C07282=1029.317,321.724,369.650,171.379,46.415,159.024
C07283=1029.324,321.936,369.619,171.383,46.415,159.025
C07284=1029.330,322.147,369.590,171.388,46.415,159.025
C07285=1029.337,322.395,369.555,171.392,46.415,159.026
C07286=1029.345,322.642,369.521,171.398,46.415,159.026
C07287=1029.351,322.890,369.486,171.403,46.416,159.027
C07288=1029.360,323.137,369.451,171.409,46.416,159.028
C07289=1029.366,323.385,369.416,171.414,46.416,159.028
C07290=1029.374,323.632,369.382,171.419,46.416,159.029
C07291=1029.381,323.879,369.348,171.424,46.416,159.030
C07292=1029.388,324.127,369.312,171.429,46.416,159.030
C07293=1029.396,324.375,369.278,171.435,46.417,159.031
C07294=1029.403,324.622,369.243,171.441,46.417,159.032
C07295=1029.410,324.869,369.208,171.445,46.417,159.032
C07296=1029.418,325.117,369.173,171.451,46.417,159.033
C07297=1029.425,325.364,369.138,171.457,46.417,159.034
C07298=1029.433,325.611,369.104,171.461,46.417,159.034
C07299=1029.440,325.859,369.068,171.467,46.417,159.035
C07300=1029.447,326.106,369.034,171.473,46.418,159.036
C07301=1029.455,326.354,368.998,171.478,46.418,159.037
C07302=1029.462,326.601,368.964,171.483,46.418,159.037
C07303=1029.470,326.848,368.929,171.489,46.419,159.038
C07304=1029.477,327.096,368.894,171.494,46.419,159.039
C07305=1029.485,327.344,368.859,171.499,46.419,159.039
C07306=1029.492,327.592,368.823,171.505,46.419,159.040
C07307=1029.500,327.839,368.789,171.510,46.420,159.041
C07308=1029.506,328.086,368.754,171.516,46.420,159.042
C07309=1029.514,328.333,368.718,171.521,46.420,159.042
C07310=1029.521,328.581,368.682,171.526,46.421,159.043
C07311=1029.528,328.828,368.647,171.532,46.421,159.044
C07312=1029.535,329.076,368.611,171.538,46.421,159.044
C07313=1029.543,329.323,368.577,171.543,46.422,159.045
C07314=1029.550,329.571,368.541,171.548,46.422,159.046
C07315=1029.557,329.817,368.505,171.554,46.423,159.047
C07316=1029.565,330.066,368.470,171.559,46.423,159.047
C07317=1029.572,330.312,368.434,171.565,46.423,159.048
C07318=1029.578,330.560,368.399,171.571,46.424,159.049
C07319=1029.586,330.807,368.362,171.576,46.425,159.050
C07320=1029.594,331.054,368.328,171.581,46.425,159.050
C07321=1029.601,331.302,368.292,171.587,46.425,159.051
C07322=1029.608,331.549,368.257,171.593,46.426,159.052
C07323=1029.616,331.796,368.220,171.598,46.427,159.053
C07324=1029.623,332.045,368.185,171.604,46.426,159.053
C07325=1029.630,332.291,368.149,171.610,46.427,159.054
C07326=1029.638,332.539,368.113,171.615,46.428,159.055
C07327=1029.645,332.786,368.078,171.620,46.428,159.056
C07328=1029.653,333.033,368.042,171.626,46.429,159.057
C07329=1029.660,333.280,368.006,171.632,46.429,159.058
C07330=1029.667,333.528,367.971,171.638,46.429,159.058
C07331=1029.675,333.775,367.934,171.643,46.430,159.059
C07332=1029.682,334.022,367.899,171.649,46.431,159.060
C07333=1029.690,334.270,367.863,171.655,46.431,159.061
C07334=1029.697,334.518,367.827,171.660,46.432,159.061
C07335=1029.704,334.764,367.791,171.665,46.433,159.062
C07336=1029.712,335.012,367.755,171.671,46.433,159.063
C07337=1029.718,335.222,367.724,171.676,46.434,159.064
C07338=1029.724,335.431,367.693,171.681,46.434,159.064
C07339=1029.730,335.641,367.663,171.686,46.435,159.065
C07340=1029.737,335.849,367.632,171.690,46.435,159.066
C07341=1029.743,336.059,367.602,171.695,46.436,159.067
C07342=1029.749,336.269,367.571,171.700,46.437,159.067
C07343=1029.756,336.478,367.541,171.706,46.437,159.068
C07344=1029.762,336.687,367.510,171.711,46.437,159.069
C07345=1029.769,336.935,367.474,171.716,46.438,159.069
C07346=1029.776,337.182,367.438,171.721,46.439,159.070
C07347=1029.784,337.429,367.400,171.727,46.439,159.071
C07348=1029.791,337.676,367.364,171.734,46.440,159.072
C07349=1029.799,337.924,367.328,171.740,46.441,159.073
C07350=1029.807,338.171,367.292,171.745,46.441,159.074
C07351=1029.814,338.418,367.256,171.750,46.442,159.075
C07352=1029.821,338.665,367.220,171.756,46.443,159.075
C07353=1029.829,338.913,367.184,171.762,46.444,159.076
C07354=1029.837,339.160,367.147,171.768,46.444,159.077
C07355=1029.844,339.407,367.110,171.774,46.445,159.078
C07356=1029.851,339.654,367.074,171.781,46.446,159.079
C07357=1029.859,339.901,367.038,171.786,46.447,159.080
C07358=1029.867,340.148,367.001,171.791,46.447,159.081
C07359=1029.874,340.396,366.965,171.798,46.449,159.082
C07360=1029.881,340.643,366.928,171.803,46.449,159.083
C07361=1029.889,340.890,366.891,171.809,46.450,159.083
C07362=1029.897,341.138,366.855,171.816,46.451,159.084
C07363=1029.904,341.385,366.817,171.822,46.451,159.085
C07364=1029.912,341.632,366.781,171.828,46.452,159.086
C07365=1029.919,341.878,366.744,171.834,46.453,159.087
C07366=1029.926,342.126,366.707,171.840,46.454,159.088
C07367=1029.934,342.373,366.671,171.846,46.455,159.089
C07368=1029.941,342.621,366.634,171.851,46.456,159.090
C07369=1029.949,342.868,366.597,171.857,46.457,159.091
C07370=1029.957,343.114,366.560,171.863,46.458,159.092
C07371=1029.964,343.362,366.523,171.869,46.459,159.093
C07372=1029.972,343.609,366.486,171.875,46.459,159.094
C07373=1029.979,343.856,366.449,171.881,46.461,159.095
C07374=1029.987,344.104,366.412,171.888,46.462,159.096
C07375=1029.995,344.350,366.375,171.894,46.462,159.096
C07376=1030.002,344.598,366.338,171.900,46.463,159.097
C07377=1030.010,344.844,366.301,171.906,46.464,159.098
C07378=1030.017,345.092,366.264,171.912,46.466,159.099
C07379=1030.026,345.340,366.227,171.918,46.466,159.100
C07380=1030.033,345.587,366.189,171.924,46.467,159.101
C07381=1030.041,345.834,366.152,171.931,46.468,159.102
C07382=1030.048,346.081,366.115,171.937,46.469,159.103
C07383=1030.056,346.328,366.078,171.943,46.471,159.104
C07384=1030.063,346.575,366.040,171.949,46.471,159.105
C07385=1030.071,346.822,366.004,171.955,46.472,159.106
C07386=1030.079,347.069,365.966,171.961,46.473,159.107
C07387=1030.087,347.316,365.929,171.968,46.474,159.108
C07388=1030.094,347.563,365.891,171.974,46.476,159.109
C07389=1030.102,347.810,365.854,171.980,46.477,159.110
C07390=1030.110,348.057,365.817,171.986,46.478,159.111
C07391=1030.118,348.304,365.780,171.992,46.479,159.112
C07392=1030.125,348.552,365.742,171.999,46.480,159.113
C07393=1030.133,348.799,365.704,172.005,46.481,159.114
C07394=1030.141,349.046,365.667,172.011,46.482,159.115
C07395=1030.148,349.292,365.629,172.017,46.483,159.116
C07396=1030.156,349.540,365.591,172.024,46.484,159.117
C07397=1030.169,349.956,365.529,172.035,46.486,159.119
C07398=1030.181,350.371,365.465,172.046,46.488,159.121
C07399=1030.195,350.787,365.401,172.056,46.490,159.123
C07400=1030.208,351.203,365.338,172.067,46.492,159.124
C07401=1030.215,351.449,365.300,172.073,46.494,159.126
C07402=1030.223,351.697,365.262,172.080,46.495,159.127
C07403=1030.231,351.943,365.224,172.086,46.496,159.128
C07404=1030.239,352.191,365.187,172.092,46.497,159.129
C07405=1030.247,352.437,365.148,172.099,46.499,159.130
C07406=1030.254,352.685,365.111,172.106,46.500,159.131
C07407=1030.262,352.932,365.072,172.112,46.501,159.132
C07408=1030.271,353.178,365.035,172.119,46.503,159.133
C07409=1030.279,353.426,364.997,172.125,46.504,159.134
C07410=1030.286,353.672,364.958,172.131,46.506,159.135
C07411=1030.294,353.920,364.920,172.139,46.506,159.136
C07412=1030.301,354.167,364.882,172.145,46.508,159.138
C07413=1030.310,354.414,364.844,172.151,46.509,159.139
C07414=1030.318,354.660,364.806,172.157,46.510,159.140
C07415=1030.326,354.907,364.767,172.164,46.512,159.141
C07416=1030.333,355.154,364.730,172.172,46.514,159.142
C07417=1030.341,355.402,364.691,172.178,46.515,159.143
C07418=1030.349,355.648,364.653,172.184,46.516,159.144
C07419=1030.358,355.895,364.615,172.190,46.517,159.145
C07420=1030.365,356.142,364.577,172.198,46.519,159.146
C07421=1030.374,356.389,364.538,172.204,46.521,159.148
C07422=1030.381,356.635,364.500,172.211,46.522,159.149
C07423=1030.389,356.883,364.461,172.217,46.523,159.150
C07424=1030.397,357.130,364.423,172.225,46.525,159.151
C07425=1030.405,357.376,364.384,172.231,46.527,159.152
C07426=1030.413,357.623,364.346,172.237,46.528,159.153
C07427=1030.421,357.870,364.308,172.244,46.529,159.155
C07428=1030.429,358.117,364.269,172.252,46.531,159.156
C07429=1030.437,358.364,364.230,172.258,46.532,159.157
C07430=1030.445,358.610,364.191,172.265,46.534,159.158
C07431=1030.453,358.858,364.153,172.272,46.536,159.159
C07432=1030.461,359.105,364.114,172.278,46.537,159.160
C07433=1030.469,359.352,364.076,172.285,46.538,159.162
C07434=1030.477,359.598,364.037,172.292,46.540,159.163
C07435=1030.485,359.845,363.998,172.299,46.542,159.164
C07436=1030.493,360.092,363.959,172.305,46.543,159.165
C07437=1030.502,360.339,363.920,172.313,46.545,159.167
C07438=1030.509,360.586,363.881,172.319,46.546,159.168
C07439=1030.517,360.832,363.842,172.326,46.548,159.169
C07440=1030.525,361.080,363.803,172.333,46.549,159.170
C07441=1030.534,361.326,363.764,172.340,46.552,159.172
C07442=1030.542,361.573,363.725,172.347,46.553,159.173
C07443=1030.549,361.820,363.686,172.354,46.555,159.174
C07444=1030.557,362.067,363.647,172.361,46.557,159.175
C07445=1030.566,362.313,363.608,172.369,46.559,159.177
C07446=1030.573,362.560,363.568,172.375,46.560,159.178
C07447=1030.582,362.807,363.529,172.382,46.562,159.179
C07448=1030.590,363.054,363.490,172.389,46.563,159.180
C07449=1030.598,363.300,363.451,172.396,46.566,159.182
C07450=1030.606,363.547,363.411,172.404,46.567,159.183
C07451=1030.614,363.794,363.373,172.410,46.569,159.184
C07452=1030.622,364.041,363.333,172.418,46.571,159.186
C07453=1030.629,364.252,363.299,172.423,46.572,159.187
C07454=1030.637,364.463,363.265,172.430,46.574,159.188
C07455=1030.643,364.673,363.232,172.436,46.575,159.189
C07456=1030.650,364.884,363.198,172.441,46.577,159.190
C07457=1030.657,365.096,363.164,172.448,46.578,159.191
C07458=1030.665,365.307,363.131,172.454,46.580,159.192
C07459=1030.671,365.518,363.097,172.460,46.582,159.194
C07460=1030.678,365.729,363.063,172.466,46.583,159.195
C07461=1030.686,365.976,363.024,172.474,46.585,159.196
C07462=1030.694,366.222,362.984,172.480,46.587,159.197
C07463=1030.703,366.468,362.944,172.488,46.589,159.199
C07464=1030.711,366.715,362.904,172.495,46.591,159.200
C07465=1030.719,366.962,362.865,172.503,46.592,159.201
C07466=1030.728,367.209,362.825,172.509,46.595,159.203
C07467=1030.736,367.456,362.785,172.517,46.597,159.204
C07468=1030.745,367.703,362.746,172.525,46.598,159.205
C07469=1030.753,367.949,362.707,172.532,46.600,159.207
C07470=1030.761,368.195,362.666,172.539,46.602,159.208
C07471=1030.770,368.442,362.627,172.546,46.605,159.210
C07472=1030.779,368.689,362.587,172.554,46.606,159.211
C07473=1030.787,368.936,362.546,172.562,46.608,159.212
C07474=1030.795,369.182,362.507,172.569,46.610,159.214
C07475=1030.803,369.429,362.467,172.576,46.612,159.215
C07476=1030.812,369.675,362.427,172.583,46.615,159.217
C07477=1030.820,369.923,362.387,172.591,46.617,159.218
C07478=1030.828,370.169,362.346,172.599,46.619,159.219
C07479=1030.837,370.415,362.306,172.606,46.621,159.221
C07480=1030.844,370.662,362.266,172.613,46.623,159.222
C07481=1030.853,370.909,362.225,172.621,46.625,159.224
C07482=1030.862,371.155,362.185,172.628,46.627,159.225
C07483=1030.870,371.402,362.145,172.636,46.629,159.227
C07484=1030.878,371.649,362.104,172.644,46.632,159.228
C07485=1030.887,371.895,362.064,172.651,46.634,159.230
C07486=1030.895,372.142,362.024,172.659,46.636,159.231
C07487=1030.903,372.389,361.983,172.667,46.638,159.232
C07488=1030.912,372.635,361.943,172.674,46.640,159.234
C07489=1030.920,372.881,361.903,172.682,46.643,159.235
C07490=1030.929,373.128,361.862,172.689,46.645,159.237
C07491=1030.937,373.374,361.822,172.697,46.646,159.238
C07492=1030.946,373.621,361.781,172.705,46.649,159.240
C07493=1030.954,373.867,361.740,172.712,46.651,159.241
C07494=1030.963,374.113,361.700,172.720,46.653,159.243
C07495=1030.972,374.360,361.659,172.728,46.656,159.244
C07496=1030.980,374.606,361.618,172.736,46.658,159.246
C07497=1030.989,374.853,361.578,172.743,46.661,159.248
C07498=1030.997,375.099,361.537,172.751,46.663,159.249
C07499=1031.006,375.346,361.496,172.759,46.665,159.251
C07500=1031.015,375.593,361.456,172.767,46.667,159.252
C07501=1031.023,375.839,361.415,172.775,46.670,159.254
C07502=1031.032,376.086,361.373,172.783,46.672,159.255
C07503=1031.041,376.332,361.333,172.791,46.674,159.257
C07504=1031.049,376.578,361.292,172.798,46.677,159.258
C07505=1031.058,376.825,361.251,172.806,46.679,159.260
C07506=1031.067,377.071,361.211,172.814,46.681,159.261
C07507=1031.076,377.318,361.170,172.822,46.684,159.263
C07508=1031.085,377.564,361.128,172.830,46.686,159.265
C07509=1031.093,377.810,361.087,172.838,46.688,159.266
C07510=1031.102,378.057,361.046,172.846,46.691,159.268
C07511=1031.110,378.304,361.005,172.855,46.694,159.269
C07512=1031.118,378.549,360.963,172.863,46.696,159.271
C07513=1031.127,378.771,360.926,172.870,46.698,159.272
C07514=1031.135,378.992,360.889,172.877,46.701,159.274
C07515=1031.142,379.214,360.852,172.885,46.703,159.276
C07516=1031.150,379.436,360.815,172.891,46.705,159.277
C07517=1031.158,379.657,360.778,172.899,46.708,159.279
C07518=1031.165,379.879,360.740,172.906,46.710,159.280
C07519=1031.173,380.100,360.703,172.913,46.712,159.281
C07520=1031.181,380.322,360.666,172.921,46.715,159.283
C07521=1031.190,380.568,360.624,172.930,46.717,159.285
C07522=1031.199,380.814,360.583,172.938,46.720,159.286
C07523=1031.207,381.060,360.541,172.946,46.722,159.288
C07524=1031.216,381.307,360.499,172.954,46.725,159.290
C07525=1031.225,381.553,360.457,172.962,46.728,159.291
C07526=1031.234,381.799,360.415,172.971,46.730,159.293
C07527=1031.242,382.046,360.374,172.979,46.733,159.295
C07528=1031.251,382.292,360.332,172.987,46.736,159.297
C07529=1031.260,382.539,360.290,172.995,46.739,159.298
C07530=1031.269,382.785,360.249,173.004,46.741,159.300
C07531=1031.278,383.031,360.207,173.012,46.744,159.302
C07532=1031.287,383.277,360.164,173.020,46.747,159.303
C07533=1031.296,383.523,360.123,173.030,46.750,159.305
C07534=1031.305,383.770,360.081,173.038,46.752,159.307
C07535=1031.314,384.016,360.039,173.046,46.755,159.309
C07536=1031.323,384.262,359.997,173.054,46.758,159.310
C07537=1031.332,384.508,359.955,173.063,46.761,159.312
C07538=1031.341,384.755,359.913,173.072,46.764,159.314
C07539=1031.351,385.000,359.871,173.080,46.766,159.316
C07540=1031.360,385.247,359.829,173.089,46.769,159.318
C07541=1031.369,385.493,359.786,173.097,46.772,159.319
C07542=1031.378,385.740,359.745,173.106,46.775,159.321
C07543=1031.387,385.986,359.703,173.115,46.778,159.323
C07544=1031.396,386.232,359.661,173.124,46.781,159.325
C07545=1031.406,386.477,359.618,173.132,46.784,159.327
C07546=1031.415,386.725,359.575,173.141,46.786,159.328
C07547=1031.424,386.970,359.533,173.150,46.789,159.330
C07548=1031.433,387.217,359.491,173.158,46.792,159.332
C07549=1031.442,387.463,359.449,173.167,46.795,159.334
C07550=1031.451,387.709,359.405,173.176,46.798,159.336
C07551=1031.460,387.955,359.363,173.184,46.801,159.338
C07552=1031.470,388.201,359.321,173.193,46.804,159.339
C07553=1031.479,388.448,359.277,173.203,46.807,159.341
C07554=1031.488,388.693,359.235,173.211,46.810,159.343
C07555=1031.497,388.939,359.192,173.220,46.814,159.345
C07556=1031.507,389.186,359.150,173.229,46.816,159.347
C07557=1031.515,389.432,359.107,173.238,46.819,159.349
C07558=1031.525,389.677,359.064,173.247,46.823,159.351
C07559=1031.535,389.924,359.021,173.256,46.826,159.353
C07560=1031.543,390.170,358.978,173.265,46.829,159.355
C07561=1031.553,390.416,358.935,173.274,46.832,159.357
C07562=1031.561,390.662,358.892,173.283,46.835,159.359
C07563=1031.571,390.908,358.849,173.292,46.838,159.360
C07564=1031.580,391.154,358.806,173.301,46.842,159.363
C07565=1031.589,391.400,358.763,173.310,46.844,159.364
C07566=1031.599,391.646,358.719,173.319,46.848,159.366
C07567=1031.608,391.892,358.677,173.329,46.851,159.369
C07568=1031.617,392.139,358.634,173.337,46.854,159.370
C07569=1031.627,392.384,358.590,173.347,46.858,159.372
C07570=1031.636,392.630,358.547,173.356,46.861,159.375
C07571=1031.646,392.876,358.504,173.366,46.864,159.376
C07572=1031.655,393.122,358.460,173.374,46.868,159.378
C07573=1031.665,393.362,358.418,173.384,46.870,159.380
C07574=1031.674,393.601,358.376,173.393,46.874,159.382
C07575=1031.682,393.840,358.334,173.402,46.877,159.384
C07576=1031.691,394.079,358.292,173.411,46.880,159.386
C07577=1031.701,394.318,358.248,173.421,46.884,159.388
C07578=1031.710,394.557,358.206,173.429,46.887,159.390
C07579=1031.719,394.796,358.164,173.438,46.890,159.392
C07580=1031.728,395.035,358.121,173.448,46.894,159.394
C07581=1031.738,395.281,358.078,173.458,46.897,159.397
C07582=1031.748,395.527,358.034,173.466,46.901,159.399
C07583=1031.757,395.773,357.990,173.476,46.904,159.401
C07584=1031.767,396.019,357.946,173.486,46.908,159.403
C07585=1031.776,396.264,357.902,173.495,46.911,159.405
C07586=1031.785,396.511,357.858,173.505,46.915,159.407
C07587=1031.796,396.756,357.815,173.515,46.918,159.409
C07588=1031.805,397.003,357.771,173.525,46.922,159.411
C07589=1031.815,397.248,357.726,173.534,46.926,159.414
C07590=1031.825,397.494,357.682,173.543,46.929,159.416
C07591=1031.834,397.740,357.638,173.554,46.933,159.418
C07592=1031.844,397.986,357.594,173.563,46.936,159.420
C07593=1031.853,398.232,357.549,173.573,46.940,159.422
C07594=1031.864,398.477,357.506,173.583,46.943,159.424
C07595=1031.873,398.724,357.462,173.592,46.947,159.427
C07596=1031.883,398.969,357.417,173.602,46.951,159.429
C07597=1031.893,399.215,357.373,173.612,46.954,159.431
C07598=1031.903,399.460,357.329,173.622,46.958,159.433
C07599=1031.912,399.707,357.284,173.632,46.962,159.435
C07600=1031.922,399.952,357.240,173.642,46.965,159.438
C07601=1031.931,400.198,357.195,173.653,46.969,159.440
C07602=1031.941,400.444,357.151,173.663,46.973,159.442
C07603=1031.951,400.689,357.106,173.672,46.976,159.444
C07604=1031.962,400.935,357.061,173.683,46.980,159.447
C07605=1031.971,401.181,357.016,173.693,46.984,159.449
C07606=1031.981,401.426,356.972,173.703,46.988,159.451
C07607=1031.991,401.672,356.927,173.713,46.992,159.454
C07608=1032.000,401.918,356.883,173.723,46.996,159.456
C07609=1032.010,402.164,356.838,173.733,46.999,159.458
C07610=1032.020,402.410,356.793,173.744,47.004,159.461
C07611=1032.030,402.655,356.748,173.754,47.008,159.463
C07612=1032.041,402.901,356.702,173.764,47.012,159.465
C07613=1032.050,403.146,356.657,173.774,47.015,159.468
C07614=1032.060,403.392,356.612,173.785,47.020,159.470
C07615=1032.070,403.638,356.567,173.795,47.024,159.472
C07616=1032.080,403.883,356.521,173.805,47.027,159.475
C07617=1032.089,404.129,356.476,173.815,47.032,159.477
C07618=1032.100,404.375,356.431,173.826,47.035,159.480
C07619=1032.110,404.620,356.385,173.837,47.040,159.482
C07620=1032.120,404.866,356.340,173.847,47.043,159.484
C07621=1032.130,405.111,356.295,173.858,47.048,159.487
C07622=1032.140,405.357,356.250,173.868,47.052,159.489
C07623=1032.150,405.603,356.205,173.879,47.056,159.492
C07624=1032.160,405.848,356.158,173.890,47.060,159.494
C07625=1032.170,406.093,356.113,173.900,47.064,159.497
C07626=1032.180,406.340,356.067,173.910,47.068,159.499
C07627=1032.191,406.585,356.022,173.922,47.072,159.502
C07628=1032.201,406.830,355.976,173.932,47.077,159.504
C07629=1032.211,407.076,355.931,173.943,47.081,159.507
C07630=1032.222,407.322,355.885,173.954,47.085,159.509
C07631=1032.232,407.567,355.839,173.965,47.089,159.512
C07632=1032.242,407.813,355.793,173.976,47.094,159.514
C07633=1032.252,408.064,355.746,173.987,47.098,159.517
C07634=1032.263,408.314,355.699,173.998,47.103,159.520
C07635=1032.274,408.566,355.653,174.009,47.107,159.522
C07636=1032.284,408.817,355.606,174.020,47.111,159.525
C07637=1032.295,409.063,355.560,174.031,47.116,159.527
C07638=1032.306,409.308,355.514,174.043,47.120,159.530
C07639=1032.317,409.553,355.467,174.053,47.124,159.533
C07640=1032.327,409.798,355.422,174.065,47.129,159.535
C07641=1032.338,410.044,355.375,174.076,47.133,159.538
C07642=1032.348,410.290,355.329,174.087,47.137,159.540
C07643=1032.358,410.536,355.283,174.099,47.142,159.543
C07644=1032.369,410.781,355.236,174.109,47.146,159.546
C07645=1032.379,411.027,355.190,174.121,47.151,159.548
C07646=1032.390,411.272,355.143,174.132,47.156,159.551
C07647=1032.401,411.517,355.097,174.143,47.160,159.554
C07648=1032.411,411.762,355.050,174.155,47.164,159.557
C07649=1032.421,412.008,355.004,174.166,47.169,159.559
C07650=1032.432,412.253,354.957,174.178,47.174,159.562
C07651=1032.443,412.498,354.910,174.190,47.178,159.565
C07652=1032.453,412.744,354.863,174.200,47.183,159.567
C07653=1032.464,412.990,354.817,174.212,47.188,159.570
C07654=1032.474,413.235,354.770,174.224,47.192,159.573
C07655=1032.485,413.480,354.723,174.236,47.197,159.576
C07656=1032.495,413.725,354.676,174.248,47.201,159.579
C07657=1032.506,413.970,354.629,174.258,47.206,159.581
C07658=1032.517,414.216,354.582,174.270,47.211,159.584
C07659=1032.528,414.461,354.535,174.282,47.215,159.587
C07660=1032.538,414.707,354.488,174.294,47.220,159.590
C07661=1032.550,414.952,354.441,174.306,47.225,159.593
C07662=1032.560,415.198,354.394,174.318,47.229,159.595
C07663=1032.572,415.443,354.346,174.330,47.234,159.598
C07664=1032.582,415.688,354.299,174.342,47.239,159.601
C07665=1032.593,415.934,354.252,174.354,47.244,159.604
C07666=1032.604,416.179,354.205,174.366,47.249,159.607
C07667=1032.615,416.424,354.157,174.378,47.254,159.610
C07668=1032.626,416.669,354.110,174.390,47.259,159.613
C07669=1032.637,416.917,354.062,174.402,47.264,159.616
C07670=1032.649,417.165,354.013,174.414,47.268,159.619
C07671=1032.659,417.413,353.965,174.426,47.273,159.622
C07672=1032.671,417.660,353.917,174.439,47.279,159.625
C07673=1032.681,417.905,353.870,174.451,47.284,159.628
C07674=1032.692,418.151,353.821,174.464,47.289,159.631
C07675=1032.703,418.396,353.773,174.476,47.294,159.634
C07676=1032.715,418.640,353.726,174.489,47.299,159.637
C07677=1032.726,418.886,353.677,174.501,47.304,159.640
C07678=1032.737,419.131,353.629,174.513,47.309,159.643
C07679=1032.748,419.377,353.581,174.526,47.314,159.646
C07680=1032.759,419.621,353.533,174.539,47.319,159.649
C07681=1032.770,419.866,353.485,174.551,47.324,159.652
C07682=1032.781,420.112,353.437,174.563,47.329,159.655
C07683=1032.792,420.357,353.389,174.576,47.335,159.658
C07684=1032.804,420.602,353.341,174.589,47.340,159.661
C07685=1032.815,420.847,353.293,174.602,47.345,159.665
C07686=1032.827,421.092,353.244,174.614,47.350,159.668
C07687=1032.838,421.338,353.195,174.627,47.356,159.671
C07688=1032.850,421.582,353.147,174.640,47.361,159.674
C07689=1032.861,421.827,353.099,174.653,47.366,159.677
C07690=1032.872,422.073,353.050,174.666,47.371,159.680
C07691=1032.884,422.317,353.001,174.679,47.377,159.683
C07692=1032.895,422.563,352.953,174.692,47.382,159.687
C07693=1032.907,422.826,352.901,174.706,47.388,159.690
C07694=1032.920,423.089,352.848,174.720,47.394,159.694
C07695=1032.932,423.353,352.796,174.735,47.399,159.697
C07696=1032.945,423.616,352.742,174.749,47.405,159.701
C07697=1032.956,423.861,352.693,174.761,47.411,159.704
C07698=1032.967,424.106,352.645,174.775,47.416,159.707
C07699=1032.979,424.351,352.596,174.789,47.422,159.711
C07700=1032.990,424.595,352.546,174.802,47.427,159.714
C07701=1033.002,424.841,352.497,174.815,47.433,159.717
C07702=1033.014,425.085,352.448,174.829,47.438,159.721
C07703=1033.025,425.330,352.399,174.843,47.444,159.724
C07704=1033.038,425.575,352.350,174.856,47.449,159.727
C07705=1033.049,425.820,352.301,174.870,47.455,159.731
C07706=1033.062,426.065,352.251,174.883,47.461,159.734
C07707=1033.073,426.310,352.202,174.896,47.466,159.738
C07708=1033.085,426.554,352.152,174.910,47.472,159.741
C07709=1033.096,426.800,352.102,174.924,47.478,159.745
C07710=1033.108,427.045,352.053,174.938,47.484,159.748
C07711=1033.120,427.289,352.003,174.952,47.489,159.752
C07712=1033.132,427.534,351.953,174.966,47.495,159.755
C07713=1033.143,427.779,351.904,174.980,47.501,159.758
C07714=1033.156,428.023,351.854,174.994,47.507,159.762
C07715=1033.167,428.269,351.803,175.008,47.513,159.766
C07716=1033.179,428.513,351.753,175.022,47.518,159.769
C07717=1033.191,428.758,351.703,175.036,47.525,159.773
C07718=1033.204,429.002,351.653,175.051,47.530,159.776
C07719=1033.215,429.247,351.603,175.065,47.536,159.780
C07720=1033.227,429.492,351.553,175.079,47.542,159.784
C07721=1033.239,429.736,351.503,175.093,47.548,159.787
C07722=1033.251,429.981,351.453,175.108,47.554,159.791
C07723=1033.263,430.226,351.401,175.123,47.560,159.795
C07724=1033.275,430.470,351.352,175.137,47.566,159.798
C07725=1033.287,430.715,351.301,175.151,47.572,159.802
C07726=1033.300,430.959,351.251,175.166,47.578,159.806
C07727=1033.312,431.204,351.201,175.180,47.584,159.809
C07728=1033.324,431.448,351.149,175.195,47.590,159.813
C07729=1033.336,431.693,351.099,175.210,47.596,159.817
C07730=1033.349,431.937,351.048,175.225,47.603,159.821
C07731=1033.362,432.181,350.997,175.240,47.609,159.824
C07732=1033.373,432.427,350.947,175.255,47.615,159.828
C07733=1033.386,432.671,350.896,175.269,47.621,159.832
C07734=1033.399,432.916,350.845,175.285,47.627,159.836
C07735=1033.412,433.160,350.794,175.300,47.634,159.840
C07736=1033.424,433.404,350.743,175.315,47.640,159.843
C07737=1033.436,433.649,350.692,175.330,47.646,159.847
C07738=1033.449,433.894,350.641,175.345,47.652,159.851
C07739=1033.462,434.138,350.590,175.360,47.659,159.855
C07740=1033.474,434.382,350.538,175.376,47.665,159.859
C07741=1033.487,434.627,350.487,175.391,47.671,159.863
C07742=1033.499,434.872,350.436,175.407,47.678,159.867
C07743=1033.512,435.115,350.384,175.422,47.684,159.871
C07744=1033.525,435.360,350.333,175.438,47.690,159.875
C07745=1033.537,435.604,350.281,175.453,47.697,159.879
C07746=1033.551,435.849,350.230,175.469,47.704,159.883
C07747=1033.563,436.093,350.178,175.484,47.710,159.887
C07748=1033.576,436.337,350.126,175.500,47.717,159.891
C07749=1033.588,436.582,350.074,175.516,47.723,159.895
C07750=1033.602,436.826,350.022,175.533,47.730,159.899
C07751=1033.614,437.070,349.970,175.548,47.736,159.903
C07752=1033.627,437.314,349.918,175.564,47.743,159.908
C07753=1033.641,437.569,349.864,175.581,47.750,159.912
C07754=1033.654,437.824,349.810,175.598,47.757,159.916
C07755=1033.668,438.080,349.755,175.615,47.764,159.921
C07756=1033.682,438.335,349.700,175.631,47.771,159.925
C07757=1033.694,438.580,349.648,175.648,47.778,159.929
C07758=1033.708,438.824,349.596,175.664,47.784,159.934
C07759=1033.720,439.067,349.543,175.680,47.791,159.938
C07760=1033.734,439.311,349.491,175.697,47.798,159.942
C07761=1033.747,439.555,349.438,175.714,47.805,159.946
C07762=1033.760,439.800,349.386,175.731,47.811,159.951
C07763=1033.774,440.044,349.333,175.747,47.819,159.955
C07764=1033.786,440.288,349.280,175.764,47.825,159.959
C07765=1033.800,440.532,349.227,175.780,47.832,159.964
C07766=1033.813,440.776,349.175,175.798,47.839,159.968
C07767=1033.826,441.020,349.121,175.815,47.846,159.973
C07768=1033.840,441.264,349.068,175.831,47.854,159.977
C07769=1033.853,441.507,349.016,175.849,47.861,159.982
C07770=1033.867,441.752,348.962,175.866,47.867,159.986
C07771=1033.880,441.996,348.909,175.882,47.875,159.991
C07772=1033.894,442.240,348.856,175.900,47.882,159.995
C07773=1033.907,442.484,348.803,175.917,47.888,159.999
C07774=1033.921,442.728,348.750,175.935,47.896,160.004
C07775=1033.935,442.971,348.696,175.952,47.903,160.009
C07776=1033.948,443.215,348.643,175.969,47.910,160.013
C07777=1033.962,443.458,348.590,175.987,47.917,160.018
C07778=1033.976,443.701,348.536,176.005,47.924,160.023
C07779=1033.990,443.944,348.483,176.022,47.931,160.027
C07780=1034.004,444.188,348.430,176.040,47.939,160.032
C07781=1034.020,444.431,348.379,176.057,47.946,160.036
C07782=1034.036,444.675,348.327,176.076,47.952,160.041
C07783=1034.051,444.919,348.275,176.093,47.959,160.045
C07784=1034.068,445.162,348.224,176.112,47.966,160.050
C07785=1034.085,445.406,348.174,176.130,47.972,160.054
C07786=1034.103,445.650,348.123,176.148,47.979,160.059
C07787=1034.122,445.894,348.074,176.167,47.985,160.063
C07788=1034.140,446.138,348.024,176.185,47.992,160.068
C07789=1034.160,446.382,347.976,176.203,47.998,160.073
C07790=1034.179,446.626,347.927,176.222,48.004,160.077
C07791=1034.200,446.870,347.880,176.240,48.011,160.082
C07792=1034.221,447.115,347.832,176.259,48.016,160.086
C07793=1034.242,447.359,347.785,176.278,48.022,160.091
C07794=1034.263,447.603,347.738,176.297,48.029,160.095
C07795=1034.285,447.848,347.692,176.316,48.034,160.099
C07796=1034.309,448.092,347.646,176.335,48.040,160.104
C07797=1034.333,448.337,347.601,176.354,48.046,160.108
C07798=1034.356,448.582,347.555,176.373,48.051,160.113
C07799=1034.381,448.827,347.512,176.392,48.057,160.117
C07800=1034.405,449.072,347.467,176.412,48.062,160.122
C07801=1034.431,449.318,347.423,176.431,48.068,160.126
C07802=1034.457,449.563,347.380,176.451,48.073,160.130
C07803=1034.484,449.808,347.338,176.471,48.078,160.135
C07804=1034.511,450.053,347.295,176.490,48.083,160.139
C07805=1034.538,450.298,347.253,176.510,48.088,160.143
C07806=1034.567,450.543,347.212,176.530,48.093,160.148
C07807=1034.595,450.789,347.171,176.550,48.098,160.152
C07808=1034.624,451.034,347.130,176.570,48.103,160.157
C07809=1034.653,451.280,347.090,176.591,48.107,160.161
C07810=1034.685,451.525,347.050,176.611,48.112,160.165
C07811=1034.714,451.771,347.011,176.631,48.117,160.170
C07812=1034.746,452.016,346.972,176.651,48.121,160.174
C07813=1034.798,452.413,346.910,176.685,48.129,160.181
C07814=1034.851,452.809,346.849,176.718,48.136,160.188
C07815=1034.564,452.870,346.521,176.721,48.203,160.209
C07816=1034.514,452.499,346.578,176.690,48.197,160.203
C07817=1034.465,452.126,346.636,176.659,48.191,160.196
C07818=1034.434,451.881,346.674,176.638,48.186,160.192
C07819=1034.403,451.636,346.714,176.618,48.182,160.188
C07820=1034.373,451.390,346.753,176.598,48.177,160.183
C07821=1034.343,451.144,346.794,176.577,48.172,160.179
C07822=1034.313,450.899,346.834,176.557,48.168,160.175
C07823=1034.284,450.654,346.875,176.537,48.163,160.170
C07824=1034.256,450.408,346.916,176.517,48.158,160.166
C07825=1034.228,450.163,346.958,176.497,48.153,160.162
C07826=1034.201,449.917,347.000,176.477,48.148,160.157
C07827=1034.174,449.672,347.042,176.457,48.143,160.153
C07828=1034.147,449.427,347.085,176.437,48.138,160.148
C07829=1034.122,449.182,347.129,176.418,48.132,160.144
C07830=1034.096,448.938,347.172,176.398,48.127,160.140
C07831=1034.072,448.692,347.217,176.379,48.122,160.135
C07832=1034.048,448.447,347.262,176.360,48.117,160.131
C07833=1034.024,448.203,347.306,176.341,48.111,160.126
C07834=1034.001,447.958,347.353,176.322,48.105,160.122
C07835=1033.978,447.714,347.398,176.303,48.100,160.118
C07836=1033.955,447.469,347.445,176.283,48.094,160.113
C07837=1033.934,447.224,347.492,176.264,48.088,160.109
C07838=1033.913,446.979,347.539,176.245,48.082,160.104
C07839=1033.893,446.736,347.586,176.227,48.076,160.100
C07840=1033.872,446.491,347.635,176.209,48.070,160.095
C07841=1033.853,446.247,347.683,176.189,48.064,160.091
C07842=1033.834,446.004,347.732,176.171,48.058,160.086
C07843=1033.815,445.759,347.782,176.153,48.052,160.082
C07844=1033.797,445.515,347.831,176.134,48.045,160.077
C07845=1033.779,445.272,347.882,176.116,48.039,160.073
C07846=1033.762,445.027,347.933,176.098,48.032,160.068
C07847=1033.746,444.784,347.984,176.080,48.026,160.064
C07848=1033.730,444.541,348.035,176.062,48.019,160.059
C07849=1033.715,444.297,348.087,176.044,48.012,160.054
C07850=1033.700,444.054,348.139,176.027,48.005,160.050
C07851=1033.685,443.810,348.193,176.008,47.998,160.045
C07852=1033.672,443.568,348.246,175.991,47.991,160.040
C07853=1033.658,443.325,348.299,175.973,47.984,160.036
C07854=1033.644,443.081,348.352,175.956,47.977,160.031
C07855=1033.630,442.837,348.406,175.938,47.970,160.027
C07856=1033.617,442.593,348.459,175.920,47.963,160.022
C07857=1033.603,442.349,348.512,175.903,47.956,160.018
C07858=1033.589,442.105,348.565,175.886,47.949,160.013
C07859=1033.576,441.861,348.618,175.869,47.942,160.009
C07860=1033.562,441.618,348.672,175.852,47.935,160.004
C07861=1033.549,441.374,348.725,175.834,47.928,160.000
C07862=1033.536,441.129,348.777,175.817,47.921,159.995
C07863=1033.522,440.886,348.830,175.801,47.914,159.991
C07864=1033.508,440.641,348.884,175.784,47.907,159.986
C07865=1033.495,440.397,348.936,175.766,47.900,159.982
C07866=1033.481,440.153,348.989,175.750,47.893,159.978
C07867=1033.469,439.909,349.042,175.733,47.887,159.973
C07868=1033.455,439.666,349.094,175.717,47.880,159.969
C07869=1033.443,439.421,349.147,175.700,47.873,159.965
C07870=1033.430,439.177,349.200,175.683,47.866,159.960
C07871=1033.416,438.933,349.252,175.666,47.860,159.956
C07872=1033.403,438.689,349.305,175.650,47.853,159.952
C07873=1033.389,438.445,349.357,175.633,47.846,159.948
C07874=1033.376,438.188,349.412,175.617,47.839,159.943
C07875=1033.363,437.932,349.466,175.600,47.832,159.939
C07876=1033.348,437.676,349.521,175.583,47.826,159.934
C07877=1033.336,437.420,349.576,175.565,47.819,159.930
C07878=1033.322,437.175,349.628,175.550,47.812,159.926
C07879=1033.309,436.931,349.680,175.534,47.805,159.922
C07880=1033.296,436.687,349.732,175.518,47.799,159.918
C07881=1033.284,436.443,349.784,175.502,47.792,159.914
C07882=1033.271,436.198,349.835,175.486,47.786,159.910
C07883=1033.258,435.954,349.887,175.470,47.780,159.905
C07884=1033.245,435.710,349.939,175.454,47.773,159.901
C07885=1033.233,435.465,349.991,175.438,47.767,159.897
C07886=1033.220,435.222,350.042,175.424,47.760,159.893
C07887=1033.207,434.977,350.093,175.408,47.754,159.889
C07888=1033.195,434.732,350.145,175.392,47.748,159.885
C07889=1033.181,434.488,350.197,175.377,47.741,159.881
C07890=1033.169,434.243,350.248,175.361,47.735,159.877
C07891=1033.157,433.999,350.299,175.346,47.729,159.874
C07892=1033.143,433.754,350.350,175.330,47.723,159.870
C07893=1033.132,433.510,350.401,175.315,47.716,159.866
C07894=1033.119,433.266,350.452,175.300,47.710,159.862
C07895=1033.106,433.021,350.503,175.285,47.704,159.858
C07896=1033.093,432.776,350.554,175.270,47.698,159.854
C07897=1033.081,432.532,350.606,175.255,47.692,159.850
C07898=1033.069,432.287,350.656,175.240,47.686,159.847
C07899=1033.056,432.043,350.707,175.225,47.679,159.843
C07900=1033.044,431.799,350.757,175.210,47.674,159.839
C07901=1033.031,431.554,350.808,175.196,47.667,159.835
C07902=1033.019,431.309,350.859,175.180,47.662,159.832
C07903=1033.007,431.065,350.909,175.166,47.655,159.828
C07904=1032.995,430.820,350.960,175.151,47.650,159.824
C07905=1032.982,430.575,351.010,175.136,47.643,159.820
C07906=1032.970,430.331,351.060,175.122,47.638,159.817
C07907=1032.958,430.086,351.111,175.107,47.632,159.813
C07908=1032.946,429.842,351.161,175.093,47.626,159.809
C07909=1032.934,429.597,351.211,175.078,47.620,159.806
C07910=1032.922,429.352,351.261,175.064,47.614,159.802
C07911=1032.910,429.107,351.312,175.050,47.608,159.799
C07912=1032.898,428.862,351.362,175.036,47.602,159.795
C07913=1032.886,428.618,351.412,175.021,47.597,159.791
C07914=1032.874,428.373,351.462,175.007,47.591,159.788
C07915=1032.861,428.129,351.512,174.993,47.585,159.784
C07916=1032.851,427.884,351.562,174.979,47.579,159.781
C07917=1032.838,427.639,351.612,174.965,47.574,159.777
C07918=1032.826,427.395,351.662,174.951,47.568,159.774
C07919=1032.814,427.150,351.712,174.937,47.562,159.770
C07920=1032.803,426.906,351.761,174.923,47.556,159.767
C07921=1032.791,426.660,351.811,174.909,47.551,159.763
C07922=1032.778,426.415,351.861,174.895,47.546,159.760
C07923=1032.767,426.171,351.910,174.882,47.540,159.756
C07924=1032.755,425.927,351.960,174.868,47.534,159.753
C07925=1032.743,425.681,352.009,174.854,47.529,159.750
C07926=1032.732,425.436,352.058,174.840,47.523,159.746
C07927=1032.720,425.191,352.107,174.827,47.518,159.743
C07928=1032.709,424.946,352.156,174.814,47.512,159.739
C07929=1032.697,424.702,352.206,174.800,47.507,159.736
C07930=1032.685,424.457,352.255,174.786,47.501,159.733
C07931=1032.673,424.212,352.304,174.773,47.496,159.729
C07932=1032.662,423.967,352.353,174.759,47.491,159.726
C07933=1032.651,423.722,352.402,174.747,47.485,159.723
C07934=1032.638,423.457,352.455,174.731,47.479,159.719
C07935=1032.626,423.191,352.509,174.718,47.473,159.716
C07936=1032.614,422.925,352.562,174.704,47.467,159.712
C07937=1032.601,422.660,352.614,174.689,47.462,159.709
C07938=1032.589,422.413,352.663,174.676,47.456,159.705
C07939=1032.577,422.169,352.712,174.663,47.451,159.702
C07940=1032.566,421.924,352.760,174.650,47.447,159.699
C07941=1032.555,421.679,352.809,174.637,47.441,159.696
C07942=1032.543,421.434,352.857,174.623,47.436,159.693
C07943=1032.531,421.189,352.906,174.611,47.431,159.690
C07944=1032.520,420.944,352.954,174.598,47.425,159.686
C07945=1032.509,420.698,353.002,174.585,47.420,159.683
C07946=1032.498,420.453,353.050,174.573,47.415,159.680
C07947=1032.486,420.209,353.099,174.560,47.410,159.677
C07948=1032.475,419.964,353.147,174.547,47.405,159.674
C07949=1032.464,419.719,353.195,174.535,47.400,159.671
C07950=1032.453,419.473,353.243,174.522,47.395,159.668
C07951=1032.441,419.228,353.291,174.510,47.390,159.665
C07952=1032.430,418.983,353.339,174.497,47.385,159.662
C07953=1032.420,418.738,353.387,174.484,47.380,159.659
C07954=1032.409,418.493,353.436,174.472,47.374,159.656
C07955=1032.397,418.248,353.483,174.459,47.369,159.653
C07956=1032.387,418.002,353.531,174.448,47.365,159.650
C07957=1032.376,417.757,353.579,174.435,47.360,159.647
C07958=1032.364,417.512,353.627,174.422,47.355,159.644
C07959=1032.354,417.267,353.674,174.410,47.350,159.641
C07960=1032.342,417.021,353.722,174.398,47.345,159.638
C07961=1032.332,416.777,353.770,174.386,47.341,159.635
C07962=1032.320,416.531,353.817,174.374,47.335,159.632
C07963=1032.310,416.286,353.864,174.362,47.330,159.629
C07964=1032.298,416.041,353.912,174.350,47.326,159.626
C07965=1032.288,415.795,353.959,174.338,47.321,159.623
C07966=1032.277,415.550,354.006,174.326,47.316,159.620
C07967=1032.266,415.305,354.054,174.314,47.312,159.618
C07968=1032.255,415.059,354.101,174.302,47.307,159.615
C07969=1032.244,414.814,354.148,174.290,47.302,159.612
C07970=1032.233,414.569,354.195,174.278,47.298,159.609
C07971=1032.223,414.323,354.242,174.266,47.293,159.606
C07972=1032.212,414.078,354.289,174.254,47.289,159.603
C07973=1032.201,413.833,354.336,174.242,47.283,159.600
C07974=1032.190,413.587,354.383,174.230,47.279,159.598
C07975=1032.179,413.342,354.430,174.219,47.274,159.595
C07976=1032.169,413.097,354.477,174.208,47.270,159.592
C07977=1032.158,412.852,354.524,174.196,47.266,159.589
C07978=1032.148,412.605,354.571,174.184,47.261,159.587
C07979=1032.137,412.360,354.617,174.172,47.256,159.584
C07980=1032.126,412.115,354.664,174.162,47.252,159.581
C07981=1032.115,411.870,354.711,174.150,47.247,159.578
C07982=1032.106,411.624,354.758,174.138,47.243,159.576
C07983=1032.095,411.379,354.804,174.127,47.238,159.573
C07984=1032.085,411.133,354.851,174.116,47.234,159.570
C07985=1032.074,410.888,354.897,174.104,47.230,159.568
C07986=1032.063,410.643,354.943,174.093,47.225,159.565
C07987=1032.053,410.398,354.990,174.082,47.221,159.562
C07988=1032.042,410.152,355.036,174.070,47.217,159.560
C07989=1032.032,409.906,355.082,174.059,47.212,159.557
C07990=1032.021,409.661,355.128,174.048,47.208,159.554
C07991=1032.011,409.415,355.174,174.037,47.203,159.552
C07992=1032.000,409.170,355.220,174.026,47.199,159.549
C07993=1031.990,408.924,355.266,174.015,47.195,159.547
C07994=1031.979,408.669,355.315,174.004,47.191,159.544
C07995=1031.968,408.413,355.362,173.992,47.186,159.541
C07996=1031.957,408.157,355.410,173.980,47.182,159.539
C07997=1031.941,407.771,355.482,173.962,47.175,159.535
C07998=1031.924,407.395,355.552,173.946,47.169,159.531
C07999=1031.915,407.149,355.598,173.936,47.165,159.528
C08000=1031.904,406.903,355.644,173.924,47.160,159.526
C08001=1031.894,406.658,355.689,173.914,47.156,159.523
C08002=1031.884,406.412,355.735,173.903,47.153,159.521
C08003=1031.874,406.167,355.780,173.892,47.148,159.518
C08004=1031.863,405.921,355.826,173.882,47.144,159.516
C08005=1031.853,405.676,355.872,173.871,47.140,159.513
C08006=1031.843,405.431,355.917,173.860,47.136,159.511
C08007=1031.833,405.184,355.963,173.850,47.132,159.508
C08008=1031.823,404.939,356.008,173.839,47.128,159.506
C08009=1031.813,404.693,356.054,173.828,47.124,159.504
C08010=1031.803,404.448,356.098,173.818,47.120,159.501
C08011=1031.792,404.202,356.144,173.808,47.116,159.499
C08012=1031.783,403.956,356.189,173.797,47.112,159.496
C08013=1031.773,403.711,356.234,173.787,47.108,159.494
C08014=1031.762,403.465,356.280,173.776,47.105,159.492
C08015=1031.753,403.220,356.325,173.765,47.100,159.489
C08016=1031.742,402.974,356.370,173.755,47.096,159.487
C08017=1031.733,402.728,356.415,173.745,47.092,159.485
C08018=1031.724,402.482,356.460,173.735,47.089,159.482
C08019=1031.714,402.237,356.505,173.725,47.085,159.480
C08020=1031.704,401.991,356.550,173.715,47.081,159.478
C08021=1031.694,401.745,356.595,173.704,47.077,159.475
C08022=1031.683,401.500,356.639,173.694,47.073,159.473
C08023=1031.673,401.254,356.684,173.684,47.070,159.471
C08024=1031.663,401.008,356.729,173.674,47.066,159.468
C08025=1031.654,400.763,356.774,173.664,47.062,159.466
C08026=1031.644,400.516,356.818,173.654,47.058,159.464
C08027=1031.635,400.271,356.863,173.644,47.055,159.462
C08028=1031.625,400.025,356.908,173.634,47.051,159.459
C08029=1031.615,399.779,356.952,173.624,47.047,159.457
C08030=1031.604,399.533,356.997,173.614,47.044,159.455
C08031=1031.595,399.288,357.041,173.604,47.040,159.453
C08032=1031.585,399.042,357.085,173.593,47.036,159.450
C08033=1031.576,398.796,357.130,173.584,47.033,159.448
C08034=1031.565,398.550,357.174,173.573,47.029,159.446
C08035=1031.556,398.304,357.218,173.564,47.026,159.444
C08036=1031.546,398.059,357.263,173.554,47.022,159.442
C08037=1031.536,397.813,357.306,173.544,47.019,159.439
C08038=1031.527,397.567,357.350,173.534,47.015,159.437
C08039=1031.517,397.321,357.395,173.525,47.012,159.435
C08040=1031.507,397.076,357.438,173.515,47.008,159.433
C08041=1031.498,396.830,357.482,173.505,47.005,159.431
C08042=1031.489,396.584,357.527,173.495,47.001,159.429
C08043=1031.478,396.338,357.570,173.485,46.998,159.426
C08044=1031.469,396.092,357.614,173.477,46.994,159.424
C08045=1031.460,395.846,357.658,173.467,46.991,159.422
C08046=1031.450,395.601,357.701,173.457,46.988,159.420
C08047=1031.441,395.355,357.746,173.447,46.984,159.418
C08048=1031.431,395.108,357.790,173.438,46.981,159.416
C08049=1031.421,394.863,357.833,173.428,46.978,159.414
C08050=1031.406,394.447,357.907,173.412,46.971,159.410
C08051=1031.390,394.032,357.981,173.397,46.966,159.407
C08052=1031.374,393.617,358.054,173.380,46.961,159.403
C08053=1031.358,393.202,358.128,173.365,46.955,159.400
C08054=1031.348,392.955,358.171,173.355,46.952,159.398
C08055=1031.339,392.710,358.214,173.346,46.949,159.396
C08056=1031.329,392.464,358.258,173.337,46.945,159.394
C08057=1031.319,392.218,358.301,173.328,46.942,159.392
C08058=1031.311,391.972,358.344,173.318,46.939,159.390
C08059=1031.301,391.726,358.387,173.310,46.936,159.388
C08060=1031.292,391.480,358.430,173.300,46.933,159.386
C08061=1031.282,391.234,358.474,173.290,46.930,159.384
C08062=1031.274,390.988,358.517,173.282,46.926,159.382
C08063=1031.264,390.741,358.560,173.272,46.924,159.380
C08064=1031.255,390.496,358.603,173.263,46.920,159.378
C08065=1031.246,390.250,358.646,173.255,46.917,159.376
C08066=1031.237,390.003,358.689,173.245,46.914,159.374
C08067=1031.227,389.758,358.732,173.237,46.911,159.373
C08068=1031.217,389.511,358.774,173.227,46.908,159.370
C08069=1031.209,389.265,358.817,173.219,46.905,159.369
C08070=1031.199,389.019,358.860,173.209,46.902,159.367
C08071=1031.190,388.773,358.903,173.201,46.899,159.365
C08072=1031.181,388.527,358.946,173.191,46.896,159.363
C08073=1031.172,388.280,358.988,173.183,46.893,159.361
C08074=1031.162,388.035,359.031,173.174,46.890,159.359
C08075=1031.154,387.789,359.074,173.165,46.887,159.357
C08076=1031.145,387.543,359.116,173.156,46.884,159.355
C08077=1031.135,387.296,359.158,173.148,46.881,159.354
C08078=1031.126,387.050,359.201,173.138,46.878,159.352
C08079=1031.117,386.804,359.244,173.130,46.875,159.350
C08080=1031.108,386.558,359.286,173.121,46.873,159.348
C08081=1031.099,386.311,359.328,173.112,46.870,159.346
C08082=1031.090,386.065,359.370,173.104,46.867,159.344
C08083=1031.080,385.819,359.413,173.095,46.864,159.343
C08084=1031.071,385.573,359.454,173.086,46.862,159.341
C08085=1031.062,385.327,359.497,173.077,46.858,159.339
C08086=1031.053,385.080,359.539,173.069,46.856,159.337
C08087=1031.043,384.834,359.581,173.060,46.853,159.335
C08088=1031.034,384.588,359.623,173.051,46.850,159.334
C08089=1031.026,384.341,359.665,173.043,46.848,159.332
C08090=1031.016,384.096,359.707,173.035,46.845,159.330
C08091=1031.007,383.849,359.749,173.026,46.842,159.328
C08092=1030.998,383.603,359.790,173.017,46.840,159.327
C08093=1030.990,383.357,359.832,173.009,46.837,159.325
C08094=1030.980,383.111,359.875,173.001,46.834,159.323
C08095=1030.971,382.865,359.916,172.992,46.831,159.321
C08096=1030.962,382.618,359.958,172.984,46.829,159.320
C08097=1030.953,382.372,360.000,172.976,46.826,159.318
C08098=1030.945,382.125,360.041,172.967,46.824,159.316
C08099=1030.936,381.879,360.083,172.958,46.821,159.315
C08100=1030.927,381.632,360.126,172.950,46.818,159.313
C08101=1030.918,381.386,360.167,172.942,46.816,159.311
C08102=1030.910,381.140,360.209,172.934,46.813,159.310
C08103=1030.901,380.894,360.250,172.926,46.811,159.308
C08104=1030.892,380.648,360.292,172.917,46.808,159.306
C08105=1030.883,380.401,360.334,172.909,46.805,159.304
C08106=1030.875,380.179,360.370,172.901,46.803,159.303
C08107=1030.867,379.956,360.408,172.894,46.801,159.302
C08108=1030.859,379.734,360.446,172.886,46.799,159.300
C08109=1030.852,379.510,360.484,172.879,46.796,159.299
C08110=1030.844,379.289,360.521,172.872,46.794,159.297
C08111=1030.836,379.066,360.558,172.864,46.792,159.296
C08112=1030.828,378.843,360.596,172.857,46.789,159.294
C08113=1030.821,378.620,360.633,172.849,46.787,159.293
C08114=1030.812,378.375,360.674,172.841,46.785,159.291
C08115=1030.804,378.128,360.715,172.833,46.782,159.289
C08116=1030.795,377.881,360.757,172.825,46.780,159.288
C08117=1030.786,377.636,360.799,172.818,46.778,159.286
C08118=1030.777,377.389,360.839,172.810,46.775,159.285
C08119=1030.768,377.142,360.880,172.802,46.773,159.283
C08120=1030.759,376.896,360.922,172.794,46.771,159.282
C08121=1030.751,376.650,360.962,172.786,46.768,159.280
C08122=1030.742,376.403,361.003,172.778,46.766,159.278
C08123=1030.734,376.156,361.043,172.770,46.764,159.277
C08124=1030.725,375.910,361.085,172.762,46.762,159.275
C08125=1030.716,375.663,361.125,172.754,46.759,159.274
C08126=1030.708,375.417,361.166,172.746,46.757,159.272
C08127=1030.699,375.170,361.207,172.738,46.755,159.271
C08128=1030.690,374.924,361.247,172.730,46.753,159.269
C08129=1030.682,374.677,361.288,172.723,46.750,159.268
C08130=1030.674,374.431,361.329,172.715,46.748,159.266
C08131=1030.664,374.184,361.369,172.707,46.746,159.265
C08132=1030.656,373.938,361.410,172.699,46.743,159.263
C08133=1030.648,373.691,361.451,172.691,46.742,159.261
C08134=1030.639,373.445,361.491,172.683,46.740,159.260
C08135=1030.630,373.198,361.532,172.676,46.737,159.259
C08136=1030.622,372.952,361.573,172.668,46.735,159.257
C08137=1030.613,372.706,361.613,172.660,46.733,159.256
C08138=1030.605,372.459,361.654,172.653,46.731,159.254
C08139=1030.597,372.212,361.694,172.645,46.729,159.253
C08140=1030.588,371.966,361.734,172.638,46.727,159.251
C08141=1030.580,371.719,361.775,172.630,46.724,159.250
C08142=1030.572,371.473,361.815,172.622,46.722,159.248
C08143=1030.563,371.227,361.855,172.615,46.720,159.247
C08144=1030.555,370.979,361.895,172.607,46.718,159.245
C08145=1030.546,370.733,361.936,172.599,46.716,159.244
C08146=1030.538,370.487,361.976,172.591,46.714,159.242
C08147=1030.530,370.240,362.016,172.585,46.712,159.241
C08148=1030.521,369.993,362.056,172.577,46.710,159.240
C08149=1030.513,369.746,362.096,172.569,46.708,159.238
C08150=1030.505,369.500,362.137,172.562,46.706,159.237
C08151=1030.496,369.253,362.176,172.555,46.704,159.235
C08152=1030.488,369.006,362.217,172.547,46.702,159.234
C08153=1030.479,368.760,362.257,172.540,46.700,159.233
C08154=1030.471,368.513,362.296,172.532,46.698,159.231
C08155=1030.463,368.267,362.337,172.524,46.697,159.230
C08156=1030.454,368.020,362.376,172.518,46.694,159.228
C08157=1030.445,367.773,362.416,172.510,46.692,159.227
C08158=1030.438,367.526,362.456,172.503,46.691,159.226
C08159=1030.429,367.280,362.496,172.495,46.689,159.224
C08160=1030.420,367.034,362.535,172.488,46.687,159.223
C08161=1030.413,366.787,362.575,172.481,46.685,159.222
C08162=1030.404,366.540,362.614,172.473,46.683,159.220
C08163=1030.396,366.293,362.654,172.467,46.681,159.219
C08164=1030.388,366.047,362.693,172.459,46.679,159.218
C08165=1030.380,365.800,362.733,172.451,46.678,159.216
C08166=1030.373,365.587,362.767,172.446,46.676,159.215
C08167=1030.365,365.375,362.801,172.440,46.675,159.214
C08168=1030.359,365.163,362.835,172.433,46.673,159.213
C08169=1030.351,364.951,362.869,172.426,46.672,159.212
C08170=1030.345,364.740,362.903,172.421,46.670,159.211
C08171=1030.337,364.527,362.936,172.415,46.669,159.209
C08172=1030.330,364.316,362.970,172.408,46.667,159.208
C08173=1030.323,364.103,363.004,172.402,46.666,159.207
C08174=1030.315,363.857,363.044,172.395,46.664,159.206
C08175=1030.307,363.610,363.083,172.388,46.662,159.205
C08176=1030.298,363.363,363.122,172.381,46.661,159.203
C08177=1030.290,363.116,363.161,172.374,46.659,159.202
C08178=1030.283,362.870,363.201,172.367,46.657,159.201
C08179=1030.274,362.623,363.240,172.360,46.655,159.200
C08180=1030.266,362.376,363.279,172.353,46.654,159.198
C08181=1030.259,362.129,363.319,172.346,46.652,159.197
C08182=1030.250,361.883,363.358,172.339,46.651,159.196
C08183=1030.242,361.635,363.397,172.332,46.649,159.195
C08184=1030.235,361.389,363.436,172.324,46.648,159.193
C08185=1030.227,361.142,363.475,172.318,46.645,159.192
C08186=1030.218,360.895,363.514,172.311,46.644,159.191
C08187=1030.210,360.648,363.553,172.304,46.642,159.189
C08188=1030.202,360.402,363.592,172.297,46.641,159.188
C08189=1030.194,360.155,363.630,172.290,46.640,159.187
C08190=1030.186,359.908,363.669,172.283,46.638,159.186
C08191=1030.177,359.661,363.708,172.277,46.636,159.185
C08192=1030.169,359.414,363.747,172.269,46.635,159.184
C08193=1030.162,359.168,363.785,172.263,46.633,159.182
C08194=1030.154,358.920,363.824,172.255,46.632,159.181
C08195=1030.145,358.674,363.863,172.249,46.630,159.180
C08196=1030.138,358.427,363.901,172.242,46.629,159.179
C08197=1030.129,358.180,363.940,172.235,46.628,159.178
C08198=1030.121,357.933,363.978,172.228,46.626,159.176
C08199=1030.114,357.686,364.017,172.222,46.624,159.175
C08200=1030.106,357.439,364.055,172.215,46.624,159.174
C08201=1030.097,357.192,364.094,172.208,46.622,159.173
C08202=1030.090,356.945,364.132,172.202,46.620,159.172
C08203=1030.082,356.698,364.171,172.194,46.619,159.171
C08204=1030.074,356.452,364.209,172.188,46.618,159.169
C08205=1030.066,356.204,364.248,172.181,46.616,159.168
C08206=1030.058,355.957,364.286,172.175,46.615,159.167
C08207=1030.050,355.711,364.324,172.168,46.613,159.166
C08208=1030.042,355.463,364.363,172.161,46.612,159.165
C08209=1030.035,355.217,364.401,172.155,46.611,159.164
C08210=1030.026,354.970,364.440,172.149,46.610,159.163
C08211=1030.019,354.723,364.478,172.141,46.608,159.161
C08212=1030.010,354.476,364.515,172.135,46.607,159.160
C08213=1030.003,354.229,364.554,172.129,46.606,159.159
C08214=1029.995,353.982,364.592,172.121,46.604,159.158
C08215=1029.987,353.735,364.630,172.115,46.603,159.157
C08216=1029.979,353.488,364.668,172.108,46.602,159.156
C08217=1029.971,353.241,364.706,172.102,46.601,159.155
C08218=1029.963,352.994,364.744,172.096,46.599,159.154
C08219=1029.956,352.747,364.782,172.089,46.599,159.153
C08220=1029.947,352.501,364.820,172.082,46.597,159.152
C08221=1029.939,352.253,364.858,172.076,46.596,159.151
C08222=1029.932,352.006,364.896,172.070,46.595,159.149
C08223=1029.925,351.759,364.933,172.063,46.594,159.148
C08224=1029.916,351.512,364.971,172.056,46.592,159.147
C08225=1029.909,351.265,365.009,172.050,46.591,159.146
C08226=1029.895,350.848,365.073,172.040,46.589,159.144
C08227=1029.883,350.430,365.137,172.028,46.587,159.143
C08228=1029.869,350.012,365.201,172.017,46.585,159.141
C08229=1029.857,349.594,365.264,172.007,46.583,159.139
C08230=1029.848,349.347,365.303,172.000,46.582,159.138
C08231=1029.840,349.100,365.340,171.994,46.581,159.137
C08232=1029.833,348.853,365.377,171.987,46.580,159.136
C08233=1029.826,348.606,365.415,171.981,46.579,159.135
C08234=1029.817,348.358,365.452,171.975,46.578,159.134
C08235=1029.810,348.111,365.490,171.969,46.577,159.133
C08236=1029.802,347.864,365.527,171.963,46.576,159.132
C08237=1029.795,347.618,365.565,171.957,46.575,159.131
C08238=1029.787,347.371,365.602,171.950,46.574,159.130
C08239=1029.779,347.123,365.640,171.944,46.573,159.129
C08240=1029.771,346.876,365.677,171.937,46.572,159.128
C08241=1029.764,346.629,365.713,171.931,46.571,159.127
C08242=1029.756,346.382,365.750,171.925,46.570,159.126
C08243=1029.749,346.135,365.788,171.919,46.569,159.125
C08244=1029.741,345.888,365.825,171.912,46.568,159.124
C08245=1029.733,345.641,365.862,171.906,46.568,159.123
C08246=1029.725,345.394,365.899,171.900,46.566,159.122
C08247=1029.718,345.147,365.937,171.894,46.565,159.121
C08248=1029.710,344.899,365.974,171.888,46.565,159.120
C08249=1029.703,344.652,366.011,171.882,46.564,159.119
C08250=1029.695,344.405,366.048,171.876,46.563,159.118
C08251=1029.687,344.158,366.085,171.870,46.562,159.118
C08252=1029.679,343.911,366.122,171.863,46.561,159.116
C08253=1029.673,343.663,366.159,171.858,46.560,159.116
C08254=1029.665,343.416,366.196,171.851,46.559,159.115
C08255=1029.657,343.169,366.233,171.845,46.558,159.114
C08256=1029.650,342.922,366.270,171.839,46.558,159.113
C08257=1029.642,342.675,366.307,171.833,46.557,159.112
C08258=1029.635,342.427,366.343,171.827,46.556,159.111
C08259=1029.627,342.180,366.380,171.821,46.556,159.110
C08260=1029.619,341.934,366.417,171.815,46.554,159.109
C08261=1029.612,341.686,366.454,171.809,46.554,159.108
C08262=1029.604,341.440,366.491,171.803,46.553,159.107
C08263=1029.597,341.192,366.527,171.798,46.552,159.106
C08264=1029.590,340.944,366.564,171.792,46.551,159.105
C08265=1029.582,340.697,366.601,171.786,46.550,159.105
C08266=1029.575,340.450,366.637,171.780,46.550,159.104
C08267=1029.567,340.203,366.674,171.774,46.549,159.103
C08268=1029.559,339.955,366.711,171.768,46.548,159.102
C08269=1029.552,339.709,366.746,171.762,46.548,159.101
C08270=1029.544,339.461,366.783,171.756,46.547,159.100
C08271=1029.536,339.214,366.820,171.750,46.547,159.099
C08272=1029.529,338.967,366.856,171.744,46.545,159.098
C08273=1029.522,338.719,366.893,171.738,46.545,159.098
C08274=1029.514,338.472,366.929,171.732,46.544,159.097
C08275=1029.507,338.225,366.965,171.726,46.544,159.096
C08276=1029.499,337.978,367.001,171.721,46.543,159.095
C08277=1029.491,337.731,367.038,171.715,46.543,159.094
C08278=1029.484,337.483,367.074,171.709,46.542,159.093
C08279=1029.477,337.237,367.110,171.703,46.542,159.093
C08280=1029.470,336.989,367.147,171.697,46.540,159.092
C08281=1029.462,336.741,367.183,171.691,46.540,159.091
C08282=1029.456,336.531,367.214,171.686,46.540,159.090
C08283=1029.449,336.320,367.245,171.682,46.539,159.089
C08284=1029.443,336.110,367.275,171.677,46.539,159.089
C08285=1029.437,335.900,367.305,171.672,46.538,159.088
C08286=1029.431,335.689,367.336,171.667,46.538,159.087
C08287=1029.424,335.479,367.367,171.662,46.537,159.087
C08288=1029.418,335.268,367.398,171.657,46.537,159.086
C08289=1029.412,335.057,367.429,171.652,46.536,159.085
C08290=1029.405,334.811,367.465,171.647,46.536,159.084
C08291=1029.397,334.563,367.501,171.641,46.535,159.084
C08292=1029.390,334.315,367.537,171.635,46.534,159.083
C08293=1029.383,334.068,367.573,171.629,46.534,159.082
C08294=1029.375,333.821,367.609,171.624,46.534,159.081
C08295=1029.368,333.574,367.645,171.619,46.533,159.080
C08296=1029.360,333.326,367.680,171.613,46.533,159.080
C08297=1029.353,333.079,367.716,171.607,46.532,159.079
C08298=1029.345,332.832,367.752,171.601,46.532,159.078
C08299=1029.338,332.584,367.787,171.595,46.532,159.077
C08300=1029.331,332.338,367.823,171.590,46.531,159.077
C08301=1029.323,332.089,367.859,171.584,46.530,159.076
C08302=1029.316,331.843,367.894,171.579,46.530,159.075
C08303=1029.308,331.595,367.931,171.573,46.530,159.074
C08304=1029.301,331.347,367.966,171.567,46.529,159.073
C08305=1029.293,331.101,368.001,171.562,46.529,159.073
C08306=1029.286,330.853,368.037,171.556,46.529,159.072
C08307=1029.279,330.606,368.073,171.551,46.528,159.071
C08308=1029.272,330.359,368.108,171.545,46.528,159.070
C08309=1029.264,330.111,368.144,171.540,46.527,159.070
C08310=1029.258,329.864,368.179,171.534,46.528,159.069
C08311=1029.250,329.616,368.215,171.528,46.527,159.068
C08312=1029.242,329.369,368.250,171.523,46.526,159.067
C08313=1029.235,329.121,368.285,171.518,46.526,159.067
C08314=1029.228,328.874,368.321,171.512,46.526,159.066
C08315=1029.221,328.627,368.356,171.506,46.526,159.065
C08316=1029.214,328.379,368.392,171.501,46.525,159.064
C08317=1029.207,328.132,368.427,171.496,46.525,159.064
C08318=1029.199,327.884,368.463,171.490,46.525,159.063
C08319=1029.192,327.637,368.498,171.485,46.524,159.062
C08320=1029.185,327.390,368.533,171.480,46.524,159.062
C08321=1029.177,327.142,368.568,171.474,46.524,159.061
C08322=1029.170,326.895,368.603,171.468,46.524,159.060
C08323=1029.162,326.647,368.638,171.463,46.524,159.060
C08324=1029.155,326.400,368.672,171.458,46.524,159.059
C08325=1029.148,326.153,368.708,171.452,46.523,159.058
C08326=1029.140,325.905,368.742,171.447,46.523,159.058
C08327=1029.133,325.657,368.778,171.442,46.523,159.057
C08328=1029.125,325.410,368.812,171.436,46.523,159.056
C08329=1029.118,325.162,368.848,171.430,46.523,159.056
C08330=1029.111,324.915,368.882,171.425,46.523,159.055
C08331=1029.103,324.668,368.917,171.420,46.523,159.054
C08332=1029.096,324.420,368.952,171.414,46.523,159.054
C08333=1029.088,324.173,368.987,171.410,46.523,159.053
C08334=1029.082,323.925,369.021,171.404,46.523,159.052
C08335=1029.074,323.678,369.056,171.398,46.523,159.052
C08336=1029.066,323.430,369.091,171.394,46.522,159.051
C08337=1029.059,323.183,369.126,171.388,46.523,159.050
C08338=1029.052,322.936,369.160,171.382,46.523,159.050
C08339=1029.045,322.688,369.195,171.378,46.522,159.049
C08340=1029.038,322.441,369.229,171.372,46.522,159.048
C08341=1029.030,322.193,369.264,171.367,46.522,159.048
C08342=1029.024,321.980,369.295,171.363,46.522,159.047
C08343=1029.018,321.767,369.324,171.358,46.522,159.047
C08344=1029.011,321.555,369.353,171.354,46.522,159.046
C08345=1029.006,321.342,369.384,171.349,46.522,159.045
C08346=1028.999,321.129,369.413,171.345,46.522,159.045
C08347=1028.993,320.917,369.443,171.340,46.522,159.044
C08348=1028.987,320.704,369.472,171.336,46.522,159.044
C08349=1028.981,320.491,369.502,171.331,46.522,159.043
C08350=1028.974,320.244,369.537,171.326,46.522,159.043
C08351=1028.966,319.996,369.570,171.321,46.522,159.042
C08352=1028.960,319.749,369.606,171.315,46.522,159.042
C08353=1028.952,319.501,369.639,171.310,46.522,159.041
C08354=1028.946,319.254,369.675,171.305,46.522,159.040
C08355=1028.938,319.007,369.709,171.299,46.522,159.040
C08356=1028.931,318.759,369.743,171.295,46.522,159.039
C08357=1028.924,318.511,369.777,171.290,46.522,159.039
C08358=1028.917,318.264,369.812,171.285,46.522,159.038
C08359=1028.910,318.016,369.846,171.279,46.522,159.037
C08360=1028.903,317.769,369.881,171.275,46.522,159.037
C08361=1028.896,317.521,369.915,171.269,46.522,159.036
C08362=1028.889,317.274,369.950,171.264,46.523,159.036
C08363=1028.882,317.026,369.984,171.259,46.523,159.035
C08364=1028.875,316.778,370.017,171.253,46.523,159.034
C08365=1028.868,316.531,370.053,171.249,46.522,159.034
C08366=1028.861,316.283,370.086,171.243,46.523,159.033
C08367=1028.853,316.036,370.120,171.239,46.523,159.033
C08368=1028.847,315.788,370.155,171.233,46.523,159.032
C08369=1028.840,315.541,370.189,171.229,46.523,159.031
C08370=1028.833,315.294,370.223,171.223,46.524,159.031
C08371=1028.826,315.046,370.257,171.219,46.523,159.030
C08372=1028.819,314.799,370.292,171.213,46.523,159.030
C08373=1028.812,314.551,370.325,171.209,46.524,159.029
C08374=1028.805,314.303,370.360,171.203,46.524,159.029
C08375=1028.798,314.055,370.394,171.198,46.524,159.028
C08376=1028.791,313.808,370.427,171.194,46.524,159.028
C08377=1028.785,313.561,370.462,171.188,46.524,159.027
C08378=1028.778,313.313,370.496,171.184,46.524,159.026
C08379=1028.771,313.065,370.530,171.179,46.525,159.026
C08380=1028.764,312.818,370.564,171.174,46.524,159.025
C08381=1028.757,312.571,370.598,171.169,46.525,159.025
C08382=1028.751,312.323,370.632,171.164,46.525,159.024
C08383=1028.744,312.075,370.666,171.158,46.525,159.023
C08384=1028.736,311.827,370.700,171.154,46.525,159.023
C08385=1028.730,311.580,370.733,171.149,46.525,159.022
C08386=1028.723,311.332,370.768,171.144,46.526,159.022
C08387=1028.716,311.085,370.802,171.139,46.526,159.021
C08388=1028.710,310.838,370.835,171.134,46.526,159.021
C08389=1028.702,310.590,370.869,171.130,46.527,159.020
C08390=1028.695,310.342,370.903,171.124,46.527,159.020
C08391=1028.687,310.094,370.935,171.120,46.527,159.019
C08392=1028.681,309.847,370.969,171.114,46.528,159.019
C08393=1028.674,309.600,371.002,171.110,46.528,159.018
C08394=1028.667,309.351,371.036,171.104,46.528,159.018
C08395=1028.659,309.104,371.069,171.100,46.529,159.017
C08396=1028.652,308.857,371.102,171.095,46.530,159.017
C08397=1028.645,308.609,371.135,171.091,46.530,159.016
C08398=1028.637,308.362,371.169,171.085,46.531,159.016
C08399=1028.631,308.113,371.202,171.081,46.531,159.016
C08400=1028.624,307.866,371.235,171.076,46.531,159.015
C08401=1028.617,307.619,371.269,171.071,46.532,159.014
C08402=1028.610,307.408,371.297,171.067,46.532,159.014
C08403=1028.605,307.198,371.325,171.063,46.532,159.014
C08404=1028.599,306.988,371.353,171.059,46.533,159.013
C08405=1028.592,306.778,371.381,171.055,46.533,159.013
C08406=1028.586,306.567,371.409,171.050,46.533,159.012
C08407=1028.581,306.357,371.437,171.047,46.534,159.012
C08408=1028.575,306.146,371.466,171.043,46.535,159.012
C08409=1028.569,305.937,371.493,171.039,46.535,159.011
C08410=1028.562,305.689,371.526,171.034,46.535,159.011
C08411=1028.555,305.442,371.560,171.029,46.536,159.011
C08412=1028.548,305.194,371.592,171.025,46.537,159.010
C08413=1028.540,304.946,371.626,171.019,46.537,159.010
C08414=1028.534,304.698,371.659,171.015,46.537,159.009
C08415=1028.527,304.450,371.692,171.010,46.537,159.009
C08416=1028.520,304.203,371.725,171.005,46.538,159.008
C08417=1028.513,303.955,371.758,171.001,46.539,159.008
C08418=1028.507,303.707,371.791,170.995,46.539,159.007
C08419=1028.499,303.460,371.824,170.991,46.540,159.007
C08420=1028.492,303.213,371.857,170.987,46.541,159.007
C08421=1028.486,302.964,371.890,170.982,46.541,159.006
C08422=1028.479,302.717,371.922,170.977,46.542,159.006
C08423=1028.471,302.469,371.956,170.973,46.542,159.005
C08424=1028.465,302.222,371.989,170.968,46.543,159.005
C08425=1028.457,301.974,372.021,170.963,46.543,159.004
C08426=1028.451,301.726,372.054,170.959,46.544,159.004
C08427=1028.444,301.478,372.087,170.954,46.544,159.003
C08428=1028.437,301.231,372.120,170.949,46.545,159.003
C08429=1028.430,300.983,372.153,170.945,46.545,159.003
C08430=1028.424,300.735,372.186,170.940,46.546,159.002
C08431=1028.417,300.488,372.218,170.936,46.547,159.002
C08432=1028.410,300.240,372.251,170.931,46.547,159.001
C08433=1028.404,299.992,372.284,170.926,46.548,159.001
C08434=1028.397,299.744,372.317,170.922,46.549,159.000
C08435=1028.390,299.496,372.349,170.917,46.549,159.000
C08436=1028.383,299.249,372.382,170.912,46.550,159.000
C08437=1028.376,299.001,372.415,170.908,46.551,158.999
C08438=1028.369,298.753,372.447,170.904,46.551,158.999
C08439=1028.363,298.506,372.480,170.898,46.552,158.998
C08440=1028.356,298.257,372.513,170.894,46.552,158.998
C08441=1028.349,298.010,372.545,170.890,46.553,158.998
C08442=1028.343,297.763,372.578,170.885,46.554,158.997
C08443=1028.336,297.514,372.611,170.880,46.554,158.997
C08444=1028.329,297.267,372.643,170.876,46.555,158.996
C08445=1028.323,297.019,372.676,170.872,46.556,158.996
C08446=1028.316,296.772,372.708,170.867,46.556,158.996
C08447=1028.309,296.524,372.741,170.862,46.557,158.995
C08448=1028.302,296.276,372.774,170.858,46.557,158.995
C08449=1028.296,296.028,372.806,170.854,46.558,158.995
C08450=1028.289,295.781,372.838,170.849,46.559,158.994
C08451=1028.283,295.532,372.871,170.844,46.559,158.994
C08452=1028.276,295.285,372.904,170.840,46.560,158.993
C08453=1028.269,295.038,372.936,170.836,46.561,158.993
C08454=1028.263,294.789,372.968,170.832,46.562,158.993
C08455=1028.257,294.542,373.001,170.826,46.563,158.992
C08456=1028.249,294.294,373.033,170.822,46.563,158.992
C08457=1028.243,294.046,373.066,170.818,46.564,158.992
C08458=1028.236,293.798,373.097,170.814,46.565,158.991
C08459=1028.229,293.551,373.129,170.809,46.566,158.991
C08460=1028.223,293.302,373.162,170.804,46.566,158.990
C08461=1028.216,293.055,373.194,170.800,46.567,158.990
C08462=1028.204,292.652,373.246,170.793,46.568,158.990
C08463=1028.194,292.249,373.298,170.785,46.570,158.989
C08464=1028.182,291.845,373.350,170.778,46.572,158.989
C08465=1028.172,291.441,373.402,170.771,46.573,158.988
C08466=1028.165,291.194,373.434,170.767,46.574,158.988
C08467=1028.158,290.946,373.466,170.763,46.575,158.987
C08468=1028.151,290.698,373.497,170.758,46.575,158.987
C08469=1028.144,290.450,373.530,170.754,46.577,158.987
C08470=1028.137,290.202,373.561,170.750,46.578,158.986
C08471=1028.131,289.954,373.593,170.745,46.578,158.986
C08472=1028.124,289.707,373.625,170.741,46.579,158.986
C08473=1028.117,289.459,373.657,170.736,46.580,158.985
C08474=1028.111,289.211,373.688,170.732,46.581,158.985
C08475=1028.104,288.964,373.720,170.728,46.582,158.985
C08476=1028.098,288.716,373.752,170.724,46.583,158.985
C08477=1028.091,288.468,373.784,170.719,46.584,158.984
C08478=1028.084,288.220,373.815,170.715,46.585,158.984
C08479=1028.076,287.972,373.848,170.710,46.586,158.984
C08480=1028.070,287.724,373.879,170.706,46.587,158.983
C08481=1028.063,287.476,373.911,170.702,46.588,158.983
C08482=1028.056,287.228,373.942,170.697,46.589,158.983
C08483=1028.050,286.980,373.974,170.693,46.590,158.982
C08484=1028.044,286.732,374.006,170.689,46.590,158.982
C08485=1028.037,286.484,374.037,170.685,46.592,158.982
C08486=1028.030,286.236,374.068,170.681,46.593,158.982
C08487=1028.023,285.989,374.101,170.676,46.594,158.981
C08488=1028.016,285.741,374.132,170.672,46.595,158.981
C08489=1028.010,285.493,374.163,170.668,46.596,158.981
C08490=1028.003,285.245,374.195,170.664,46.597,158.980
C08491=1027.996,284.997,374.226,170.660,46.598,158.980
C08492=1027.989,284.749,374.256,170.654,46.599,158.980
C08493=1027.982,284.501,374.288,170.650,46.600,158.980
C08494=1027.976,284.253,374.319,170.646,46.601,158.979
C08495=1027.969,284.005,374.351,170.642,46.603,158.979
C08496=1027.962,283.757,374.382,170.638,46.604,158.979
C08497=1027.955,283.509,374.414,170.634,46.605,158.979
C08498=1027.949,283.262,374.445,170.629,46.606,158.978
C08499=1027.942,283.014,374.476,170.625,46.607,158.978
C08500=1027.935,282.766,374.508,170.621,46.608,158.978
C08501=1027.928,282.518,374.538,170.617,46.609,158.978
C08502=1027.921,282.270,374.569,170.613,46.610,158.977
C08503=1027.915,282.022,374.601,170.609,46.611,158.977
C08504=1027.908,281.774,374.632,170.604,46.612,158.977
C08505=1027.902,281.526,374.663,170.600,46.614,158.977
C08506=1027.895,281.278,374.694,170.596,46.615,158.976
C08507=1027.889,281.030,374.726,170.592,46.616,158.976
C08508=1027.882,280.782,374.757,170.588,46.617,158.976
C08509=1027.875,280.534,374.787,170.584,46.618,158.976
C08510=1027.868,280.286,374.819,170.579,46.620,158.975
C08511=1027.861,280.038,374.850,170.575,46.621,158.975
C08512=1027.855,279.790,374.881,170.571,46.622,158.975
C08513=1027.849,279.543,374.912,170.567,46.623,158.975
C08514=1027.842,279.295,374.943,170.563,46.625,158.975
C08515=1027.836,279.046,374.974,170.559,46.626,158.974
C08516=1027.829,278.798,375.005,170.555,46.627,158.974
C08517=1027.821,278.551,375.036,170.551,46.628,158.974
C08518=1027.812,278.159,375.084,170.544,46.630,158.973
C08519=1027.801,277.768,375.134,170.538,46.632,158.973
C08520=1027.791,277.377,375.183,170.531,46.634,158.973
C08521=1027.780,276.986,375.231,170.525,46.636,158.972
C08522=1027.773,276.738,375.262,170.521,46.637,158.972
C08523=1027.767,276.490,375.292,170.516,46.638,158.972
C08524=1027.760,276.242,375.323,170.513,46.640,158.972
C08525=1027.753,275.994,375.354,170.509,46.641,158.972
C08526=1027.747,275.745,375.385,170.505,46.643,158.971
C08527=1027.740,275.498,375.416,170.501,46.644,158.971
C08528=1027.734,275.250,375.446,170.497,46.645,158.971
C08529=1027.727,275.002,375.476,170.493,46.646,158.971
C08530=1027.720,274.754,375.507,170.489,46.647,158.971
C08531=1027.713,274.505,375.538,170.485,46.648,158.970
C08532=1027.707,274.258,375.568,170.480,46.650,158.970
C08533=1027.700,274.009,375.599,170.476,46.651,158.970
C08534=1027.693,273.762,375.629,170.472,46.653,158.970
C08535=1027.687,273.514,375.660,170.468,46.654,158.970
C08536=1027.681,273.265,375.691,170.465,46.656,158.970
C08537=1027.674,273.017,375.721,170.460,46.657,158.969
C08538=1027.667,272.770,375.752,170.457,46.659,158.969
C08539=1027.660,272.522,375.782,170.453,46.660,158.969
C08540=1027.654,272.273,375.813,170.449,46.661,158.969
C08541=1027.647,272.026,375.842,170.445,46.662,158.969
C08542=1027.641,271.777,375.873,170.441,46.664,158.969
C08543=1027.634,271.529,375.903,170.436,46.665,158.968
C08544=1027.628,271.282,375.934,170.432,46.667,158.968
C08545=1027.620,271.034,375.964,170.428,46.668,158.968
C08546=1027.614,270.785,375.995,170.425,46.670,158.968
C08547=1027.607,270.538,376.025,170.421,46.671,158.968
C08548=1027.601,270.289,376.056,170.417,46.673,158.968
C08549=1027.594,270.041,376.086,170.413,46.674,158.967
C08550=1027.588,269.793,376.116,170.409,46.675,158.967
C08551=1027.581,269.545,376.146,170.405,46.677,158.967
C08552=1027.574,269.297,376.176,170.401,46.678,158.967
C08553=1027.568,269.049,376.207,170.397,46.680,158.967
C08554=1027.561,268.801,376.237,170.394,46.681,158.967
C08555=1027.554,268.553,376.266,170.390,46.682,158.966
C08556=1027.548,268.305,376.297,170.386,46.684,158.966
C08557=1027.541,268.056,376.327,170.381,46.686,158.966
C08558=1027.535,267.808,376.357,170.377,46.687,158.966
C08559=1027.528,267.560,376.387,170.373,46.689,158.966
C08560=1027.521,267.312,376.417,170.370,46.690,158.966
C08561=1027.515,267.064,376.448,170.366,46.692,158.966
C08562=1027.508,266.816,376.477,170.362,46.693,158.965
C08563=1027.501,266.568,376.507,170.358,46.695,158.965
C08564=1027.495,266.320,376.538,170.354,46.697,158.965
C08565=1027.489,266.071,376.567,170.351,46.698,158.965
C08566=1027.481,265.823,376.597,170.347,46.699,158.965
C08567=1027.475,265.576,376.627,170.343,46.701,158.965
C08568=1027.468,265.327,376.657,170.339,46.703,158.965
C08569=1027.462,265.079,376.687,170.335,46.704,158.965
C08570=1027.455,264.831,376.717,170.332,46.706,158.965
C08571=1027.449,264.583,376.747,170.328,46.708,158.965
C08572=1027.442,264.334,376.776,170.324,46.709,158.964
C08573=1027.435,264.087,376.806,170.320,46.711,158.964
C08574=1027.425,263.701,376.852,170.314,46.714,158.964
C08575=1027.414,263.314,376.899,170.308,46.716,158.964
C08576=1027.404,262.927,376.945,170.302,46.718,158.964
C08577=1027.394,262.541,376.991,170.297,46.721,158.964
C08578=1027.388,262.293,377.021,170.293,46.723,158.964
C08579=1027.381,262.044,377.051,170.289,46.724,158.963
C08580=1027.375,261.797,377.081,170.285,46.725,158.963
C08581=1027.368,261.548,377.110,170.281,46.727,158.963
C08582=1027.361,261.300,377.140,170.278,46.729,158.963
C08583=1027.355,261.051,377.170,170.274,46.730,158.963
C08584=1027.349,260.804,377.200,170.270,46.732,158.963
C08585=1027.342,260.556,377.228,170.265,46.734,158.963
C08586=1027.335,260.307,377.258,170.262,46.736,158.963
C08587=1027.328,260.059,377.287,170.258,46.738,158.963
C08588=1027.322,259.811,377.317,170.254,46.740,158.963
C08589=1027.315,259.563,377.346,170.251,46.742,158.963
C08590=1027.307,259.314,377.375,170.247,46.743,158.962
C08591=1027.301,259.066,377.404,170.243,46.745,158.962
C08592=1027.294,258.818,377.434,170.239,46.747,158.962
C08593=1027.288,258.570,377.463,170.236,46.748,158.962
C08594=1027.281,258.322,377.492,170.232,46.751,158.962
C08595=1027.274,258.073,377.521,170.228,46.752,158.962
C08596=1027.268,257.825,377.550,170.225,46.754,158.962
C08597=1027.260,257.577,377.580,170.221,46.756,158.962
C08598=1027.254,257.329,377.609,170.217,46.757,158.962
C08599=1027.247,257.081,377.638,170.214,46.760,158.962
C08600=1027.240,256.832,377.667,170.210,46.761,158.962
C08601=1027.234,256.584,377.696,170.206,46.763,158.962
C08602=1027.228,256.336,377.725,170.202,46.765,158.962
C08603=1027.220,256.088,377.755,170.199,46.767,158.962
C08604=1027.214,255.840,377.784,170.195,46.769,158.962
C08605=1027.207,255.592,377.813,170.192,46.771,158.962
C08606=1027.201,255.343,377.842,170.188,46.772,158.962
C08607=1027.194,255.095,377.871,170.184,46.774,158.962
C08608=1027.187,254.847,377.900,170.181,46.776,158.962
C08609=1027.181,254.598,377.929,170.177,46.778,158.962
C08610=1027.174,254.350,377.958,170.173,46.780,158.961
C08611=1027.168,254.102,377.987,170.170,46.782,158.962
C08612=1027.160,253.853,378.016,170.166,46.784,158.961
C08613=1027.154,253.605,378.045,170.162,46.785,158.961
C08614=1027.148,253.357,378.074,170.158,46.787,158.961
C08615=1027.142,253.109,378.103,170.155,46.790,158.961
C08616=1027.134,252.860,378.132,170.151,46.791,158.961
C08617=1027.128,252.612,378.161,170.147,46.793,158.961
C08618=1027.122,252.364,378.190,170.144,46.795,158.961
C08619=1027.115,252.116,378.219,170.140,46.797,158.961
C08620=1027.108,251.868,378.248,170.136,46.799,158.961
C08621=1027.102,251.619,378.277,170.133,46.801,158.961
C08622=1027.095,251.371,378.306,170.129,46.803,158.961
C08623=1027.089,251.123,378.335,170.126,46.804,158.961
C08624=1027.082,250.875,378.364,170.122,46.807,158.961
C08625=1027.075,250.627,378.393,170.118,46.808,158.961
C08626=1027.069,250.378,378.422,170.115,46.810,158.961
C08627=1027.063,250.130,378.451,170.111,46.812,158.961
C08628=1027.056,249.882,378.479,170.107,46.814,158.961
C08629=1027.050,249.634,378.508,170.104,46.817,158.961
C08630=1027.040,249.246,378.553,170.098,46.819,158.961
C08631=1027.029,248.857,378.598,170.093,46.822,158.961
C08632=1027.020,248.470,378.643,170.088,46.825,158.961
C08633=1027.009,248.082,378.688,170.082,46.828,158.961
C08634=1027.003,247.834,378.717,170.079,46.830,158.961
C08635=1026.996,247.586,378.746,170.075,46.832,158.961
C08636=1026.990,247.337,378.775,170.071,46.834,158.961
C08637=1026.983,247.089,378.803,170.068,46.836,158.961
C08638=1026.977,246.840,378.832,170.064,46.838,158.961
C08639=1026.970,246.592,378.861,170.060,46.840,158.961
C08640=1026.964,246.344,378.890,170.057,46.842,158.961
C08641=1026.957,246.096,378.918,170.053,46.844,158.961
C08642=1026.951,245.848,378.947,170.049,46.846,158.961
C08643=1026.945,245.599,378.976,170.046,46.848,158.961
C08644=1026.939,245.351,379.005,170.042,46.850,158.961
C08645=1026.932,245.103,379.033,170.040,46.852,158.961
C08646=1026.926,244.854,379.061,170.036,46.854,158.961
C08647=1026.920,244.606,379.090,170.033,46.856,158.961
C08648=1026.913,244.358,379.119,170.029,46.858,158.961
C08649=1026.907,244.109,379.147,170.025,46.860,158.961
C08650=1026.901,243.861,379.176,170.022,46.862,158.961
C08651=1026.894,243.613,379.204,170.018,46.864,158.961
C08652=1026.888,243.365,379.233,170.015,46.867,158.961
C08653=1026.881,243.116,379.261,170.011,46.868,158.961
C08654=1026.874,242.868,379.289,170.008,46.871,158.961
C08655=1026.868,242.620,379.318,170.004,46.873,158.961
C08656=1026.861,242.372,379.346,170.000,46.875,158.961
C08657=1026.855,242.122,379.375,169.998,46.877,158.961
C08658=1026.848,241.875,379.403,169.995,46.879,158.961
C08659=1026.842,241.626,379.431,169.991,46.881,158.961
C08660=1026.835,241.377,379.459,169.987,46.883,158.961
C08661=1026.829,241.129,379.488,169.984,46.886,158.961
C08662=1026.822,240.881,379.516,169.980,46.887,158.961
C08663=1026.816,240.633,379.545,169.977,46.890,158.961
C08664=1026.810,240.385,379.572,169.973,46.892,158.961
C08665=1026.803,240.137,379.600,169.970,46.894,158.961
C08666=1026.797,239.888,379.629,169.966,46.896,158.961
C08667=1026.790,239.640,379.657,169.963,46.898,158.961
C08668=1026.783,239.391,379.685,169.959,46.901,158.961
C08669=1026.777,239.143,379.712,169.956,46.903,158.962
C08670=1026.770,238.895,379.741,169.953,46.905,158.962
C08671=1026.764,238.646,379.769,169.950,46.907,158.962
C08672=1026.757,238.398,379.797,169.946,46.909,158.962
C08673=1026.750,238.150,379.825,169.943,46.912,158.962
C08674=1026.744,237.901,379.852,169.939,46.914,158.962
C08675=1026.738,237.653,379.881,169.936,46.916,158.962
C08676=1026.731,237.405,379.909,169.932,46.919,158.962
C08677=1026.724,237.156,379.937,169.929,46.921,158.962
C08678=1026.717,236.908,379.965,169.925,46.923,158.962
C08679=1026.711,236.659,379.992,169.922,46.925,158.962
C08680=1026.705,236.410,380.021,169.918,46.927,158.962
C08681=1026.698,236.162,380.048,169.915,46.930,158.962
C08682=1026.691,235.914,380.076,169.911,46.932,158.962
C08683=1026.684,235.666,380.104,169.908,46.935,158.962
C08684=1026.678,235.418,380.132,169.905,46.937,158.963
C08685=1026.672,235.170,380.160,169.902,46.939,158.963
C08686=1026.661,234.775,380.203,169.896,46.943,158.963
C08687=1026.651,234.381,380.248,169.891,46.946,158.963
C08688=1026.641,233.987,380.292,169.886,46.951,158.963
C08689=1026.630,233.592,380.336,169.881,46.954,158.963
C08690=1026.624,233.344,380.363,169.877,46.956,158.963
C08691=1026.617,233.096,380.391,169.874,46.959,158.963
C08692=1026.611,232.848,380.418,169.870,46.961,158.963
C08693=1026.605,232.599,380.447,169.867,46.964,158.963
C08694=1026.598,232.351,380.474,169.863,46.966,158.964
C08695=1026.591,232.102,380.502,169.860,46.968,158.964
C08696=1026.585,231.854,380.530,169.857,46.970,158.964
C08697=1026.578,231.605,380.558,169.854,46.973,158.964
C08698=1026.572,231.358,380.585,169.851,46.975,158.964
C08699=1026.565,231.109,380.613,169.847,46.977,158.964
C08700=1026.559,230.860,380.640,169.844,46.980,158.964
C08701=1026.552,230.612,380.667,169.840,46.982,158.964
C08702=1026.546,230.363,380.695,169.837,46.985,158.964
C08703=1026.540,230.115,380.723,169.833,46.987,158.964
C08704=1026.533,229.867,380.750,169.830,46.989,158.964
C08705=1026.526,229.618,380.777,169.826,46.992,158.965
C08706=1026.520,229.369,380.805,169.824,46.994,158.965
C08707=1026.514,229.122,380.832,169.821,46.997,158.965
C08708=1026.507,228.873,380.860,169.817,46.999,158.965
C08709=1026.501,228.624,380.887,169.814,47.001,158.965
C08710=1026.494,228.376,380.915,169.810,47.004,158.965
C08711=1026.487,228.127,380.943,169.807,47.006,158.965
C08712=1026.481,227.880,380.970,169.804,47.009,158.965
C08713=1026.475,227.631,380.997,169.800,47.012,158.966
C08714=1026.468,227.382,381.025,169.797,47.014,158.966
C08715=1026.461,227.135,381.051,169.795,47.016,158.966
C08716=1026.455,226.886,381.079,169.791,47.018,158.966
C08717=1026.448,226.637,381.106,169.788,47.021,158.966
C08718=1026.442,226.388,381.133,169.784,47.024,158.966
C08719=1026.435,226.141,381.160,169.781,47.026,158.966
C08720=1026.429,225.892,381.187,169.778,47.029,158.967
C08721=1026.422,225.643,381.215,169.774,47.032,158.967
C08722=1026.415,225.395,381.242,169.771,47.034,158.967
C08723=1026.409,225.147,381.269,169.768,47.037,158.967
C08724=1026.402,224.898,381.296,169.764,47.039,158.967
C08725=1026.396,224.649,381.323,169.761,47.042,158.967
C08726=1026.388,224.401,381.350,169.759,47.044,158.967
C08727=1026.383,224.153,381.377,169.755,47.047,158.967
C08728=1026.376,223.904,381.405,169.752,47.049,158.968
C08729=1026.369,223.655,381.431,169.749,47.052,158.968
C08730=1026.363,223.407,381.458,169.745,47.055,158.968
C08731=1026.356,223.159,381.486,169.742,47.057,158.968
C08732=1026.350,222.910,381.513,169.739,47.060,158.968
C08733=1026.343,222.662,381.539,169.735,47.062,158.968
C08734=1026.337,222.413,381.566,169.732,47.065,158.969
C08735=1026.330,222.165,381.594,169.730,47.067,158.969
C08736=1026.324,221.917,381.620,169.726,47.070,158.969
C08737=1026.317,221.668,381.647,169.723,47.073,158.969
C08738=1026.311,221.419,381.675,169.720,47.075,158.969
C08739=1026.305,221.171,381.702,169.716,47.078,158.969
C08740=1026.297,220.923,381.729,169.713,47.081,158.969
C08741=1026.292,220.674,381.755,169.710,47.083,158.969
C08742=1026.281,220.272,381.799,169.705,47.087,158.970
C08743=1026.270,219.870,381.842,169.700,47.091,158.970
C08744=1026.260,219.469,381.886,169.694,47.096,158.970
C08745=1026.250,219.067,381.930,169.689,47.100,158.971
C08746=1026.243,218.818,381.957,169.686,47.103,158.971
C08747=1026.236,218.569,381.983,169.683,47.106,158.971
C08748=1026.230,218.321,382.010,169.680,47.108,158.971
C08749=1026.223,218.073,382.037,169.677,47.111,158.971
C08750=1026.216,217.825,382.063,169.674,47.114,158.972
C08751=1026.210,217.576,382.090,169.670,47.116,158.972
C08752=1026.203,217.328,382.116,169.667,47.119,158.972
C08753=1026.197,217.079,382.143,169.664,47.122,158.972
C08754=1026.190,216.830,382.169,169.661,47.125,158.972
C08755=1026.183,216.582,382.195,169.658,47.128,158.972
C08756=1026.177,216.333,382.222,169.654,47.130,158.972
C08757=1026.170,216.085,382.249,169.651,47.133,158.973
C08758=1026.164,215.836,382.276,169.649,47.136,158.973
C08759=1026.157,215.588,382.302,169.645,47.138,158.973
C08760=1026.150,215.339,382.329,169.642,47.141,158.973
C08761=1026.144,215.090,382.356,169.639,47.144,158.974
C08762=1026.137,214.842,382.382,169.636,47.147,158.974
C08763=1026.131,214.593,382.409,169.633,47.150,158.974
C08764=1026.124,214.345,382.435,169.629,47.153,158.974
C08765=1026.118,214.096,382.462,169.626,47.155,158.974
C08766=1026.112,213.848,382.488,169.623,47.158,158.975
C08767=1026.104,213.599,382.514,169.621,47.161,158.975
C08768=1026.099,213.351,382.541,169.617,47.163,158.975
C08769=1026.092,213.102,382.567,169.614,47.166,158.975
C08770=1026.086,212.854,382.594,169.611,47.169,158.975
C08771=1026.079,212.605,382.620,169.608,47.172,158.975
C08772=1026.072,212.357,382.646,169.604,47.175,158.976
C08773=1026.066,212.109,382.673,169.601,47.178,158.976
C08774=1026.059,211.860,382.700,169.599,47.180,158.976
C08775=1026.054,211.612,382.726,169.596,47.183,158.976
C08776=1026.046,211.363,382.753,169.593,47.186,158.977
C08777=1026.040,211.115,382.779,169.589,47.189,158.977
C08778=1026.034,210.865,382.805,169.586,47.191,158.977
C08779=1026.027,210.617,382.831,169.583,47.194,158.977
C08780=1026.020,210.368,382.857,169.580,47.197,158.977
C08781=1026.014,210.120,382.884,169.578,47.200,158.978
C08782=1026.008,209.872,382.910,169.574,47.203,158.978
C08783=1026.001,209.623,382.937,169.571,47.206,158.978
C08784=1025.994,209.375,382.963,169.568,47.209,158.978
C08785=1025.987,209.126,382.988,169.565,47.212,158.979
C08786=1025.982,208.877,383.015,169.562,47.215,158.979
C08787=1025.975,208.629,383.041,169.558,47.218,158.979
C08788=1025.968,208.381,383.067,169.555,47.220,158.979
C08789=1025.962,208.132,383.093,169.552,47.223,158.979
C08790=1025.955,207.883,383.119,169.550,47.226,158.980
C08791=1025.949,207.635,383.146,169.547,47.229,158.980
C08792=1025.942,207.386,383.172,169.544,47.232,158.980
C08793=1025.936,207.137,383.198,169.540,47.235,158.980
C08794=1025.929,206.889,383.224,169.537,47.238,158.981
C08795=1025.922,206.641,383.250,169.534,47.241,158.981
C08796=1025.916,206.392,383.275,169.531,47.244,158.981
C08797=1025.909,206.143,383.302,169.528,47.247,158.981
C08798=1025.898,205.745,383.343,169.523,47.252,158.982
C08799=1025.888,205.346,383.385,169.518,47.257,158.982
C08800=1025.877,204.948,383.426,169.514,47.261,158.983
C08801=1025.867,204.549,383.468,169.508,47.267,158.983
C08802=1025.842,203.513,383.570,169.115,47.165,158.911
C08803=1025.837,203.265,383.594,169.111,47.168,158.911
C08804=1025.831,203.015,383.619,169.107,47.172,158.912
C08805=1025.825,202.767,383.643,169.103,47.176,158.912
C08806=1025.819,202.518,383.667,169.098,47.179,158.912
C08807=1025.814,202.270,383.692,169.094,47.183,158.912
C08808=1025.808,202.020,383.717,169.090,47.187,158.913
C08809=1025.802,201.772,383.740,169.086,47.191,158.913
C08810=1025.796,201.524,383.765,169.082,47.195,158.913
C08811=1025.791,201.274,383.789,169.078,47.199,158.914
C08812=1025.785,201.026,383.814,169.074,47.203,158.914
C08813=1025.779,200.776,383.838,169.071,47.207,158.914
C08814=1025.773,200.528,383.862,169.066,47.210,158.914
C08815=1025.767,200.279,383.887,169.063,47.214,158.915
C08816=1025.762,200.030,383.911,169.059,47.218,158.915
C08817=1025.756,199.782,383.934,169.055,47.222,158.915
C08818=1025.750,199.533,383.959,169.051,47.226,158.916
C08819=1025.744,199.284,383.983,169.047,47.230,158.916
C08820=1025.738,199.035,384.007,169.043,47.234,158.916
C08821=1025.732,198.787,384.031,169.039,47.238,158.917
C08822=1025.727,198.538,384.055,169.036,47.242,158.917
C08823=1025.720,198.289,384.079,169.032,47.246,158.917
C08824=1025.714,198.041,384.103,169.028,47.250,158.918
C08825=1025.709,197.791,384.127,169.024,47.254,158.918
C08826=1025.703,197.543,384.151,169.020,47.258,158.918
C08827=1025.697,197.294,384.175,169.015,47.261,158.918
C08828=1025.691,197.045,384.199,169.011,47.265,158.919
C08829=1025.685,196.797,384.223,169.007,47.269,158.919
C08830=1025.680,196.548,384.246,169.003,47.273,158.919
C08831=1025.673,196.299,384.270,168.999,47.277,158.920
C08832=1025.668,196.050,384.294,168.996,47.281,158.920
C08833=1025.662,195.802,384.318,168.992,47.285,158.920
C08834=1025.656,195.552,384.342,168.988,47.289,158.921
C08835=1025.650,195.304,384.366,168.984,47.293,158.921
C08836=1025.644,195.055,384.389,168.980,47.297,158.921
C08837=1025.638,194.806,384.414,168.976,47.301,158.922
C08838=1025.632,194.557,384.437,168.972,47.305,158.922
C08839=1025.627,194.309,384.461,168.968,47.309,158.922
C08840=1025.620,194.060,384.485,168.965,47.313,158.923
C08841=1025.615,193.810,384.509,168.961,47.317,158.923
C08842=1025.609,193.562,384.532,168.957,47.321,158.923
C08843=1025.603,193.314,384.556,168.953,47.325,158.924
C08844=1025.598,193.064,384.580,168.949,47.329,158.924
C08845=1025.592,192.816,384.603,168.946,47.333,158.924
C08846=1025.587,192.567,384.627,168.943,47.338,158.925
C08847=1025.581,192.318,384.651,168.939,47.342,158.925
C08848=1025.575,192.070,384.674,168.935,47.346,158.925
C08849=1025.569,191.820,384.698,168.931,47.350,158.926
C08850=1025.563,191.572,384.722,168.927,47.354,158.926
C08851=1025.558,191.323,384.745,168.923,47.358,158.926
C08852=1025.552,191.074,384.769,168.920,47.362,158.927
C08853=1025.546,190.825,384.792,168.916,47.366,158.927
C08854=1025.540,190.576,384.817,168.912,47.370,158.927
C08855=1025.535,190.327,384.840,168.908,47.374,158.928
C08856=1025.529,190.079,384.863,168.904,47.378,158.928
C08857=1025.524,189.830,384.887,168.900,47.382,158.928
C08858=1025.518,189.581,384.910,168.896,47.386,158.929
C08859=1025.513,189.332,384.934,168.894,47.389,158.929
C08860=1025.506,189.083,384.958,168.890,47.393,158.929
C08861=1025.500,188.834,384.981,168.886,47.397,158.930
C08862=1025.495,188.586,385.005,168.882,47.401,158.930
C08863=1025.488,188.303,385.032,168.877,47.406,158.930
C08864=1025.483,188.021,385.058,168.874,47.410,158.931
C08865=1025.476,187.738,385.085,168.869,47.415,158.931
C08866=1025.469,187.456,385.112,168.866,47.420,158.932
C08867=1025.464,187.206,385.135,168.862,47.424,158.932
C08868=1025.458,186.958,385.159,168.858,47.428,158.932
C08869=1025.452,186.709,385.182,168.854,47.432,158.933
C08870=1025.447,186.460,385.205,168.850,47.436,158.933
C08871=1025.441,186.212,385.229,168.847,47.440,158.933
C08872=1025.435,185.963,385.252,168.843,47.444,158.934
C08873=1025.430,185.714,385.276,168.840,47.448,158.934
C08874=1025.424,185.465,385.299,168.836,47.452,158.934
C08875=1025.419,185.216,385.323,168.832,47.456,158.935
C08876=1025.414,184.967,385.346,168.828,47.460,158.935
C08877=1025.407,184.718,385.370,168.825,47.464,158.935
C08878=1025.402,184.469,385.393,168.822,47.468,158.936
C08879=1025.396,184.220,385.416,168.818,47.472,158.936
C08880=1025.390,183.972,385.440,168.814,47.476,158.936
C08881=1025.385,183.723,385.463,168.810,47.480,158.937
C08882=1025.380,183.474,385.486,168.807,47.484,158.937
C08883=1025.374,183.225,385.509,168.803,47.488,158.937
C08884=1025.369,182.976,385.533,168.800,47.492,158.938
C08885=1025.363,182.727,385.557,168.796,47.496,158.938
C08886=1025.358,182.478,385.580,168.792,47.500,158.938
C08887=1025.351,182.230,385.602,168.789,47.505,158.939
C08888=1025.346,181.981,385.625,168.785,47.509,158.939
C08889=1025.340,181.732,385.648,168.782,47.513,158.940
C08890=1025.334,181.483,385.671,168.778,47.518,158.940
C08891=1025.328,181.234,385.693,168.774,47.522,158.940
C08892=1025.322,180.985,385.716,168.771,47.526,158.941
C08893=1025.317,180.736,385.739,168.767,47.530,158.941
C08894=1025.311,180.487,385.762,168.763,47.535,158.942
C08895=1025.304,180.238,385.784,168.759,47.539,158.942
C08896=1025.299,179.990,385.807,168.757,47.543,158.943
C08897=1025.293,179.741,385.830,168.753,47.547,158.943
C08898=1025.287,179.492,385.853,168.749,47.551,158.943
C08899=1025.281,179.243,385.875,168.746,47.556,158.944
C08900=1025.275,178.994,385.897,168.742,47.560,158.944
C08901=1025.270,178.745,385.920,168.738,47.565,158.944
C08902=1025.263,178.496,385.943,168.734,47.569,158.945
C08903=1025.257,178.247,385.966,168.731,47.574,158.945
C08904=1025.252,177.998,385.989,168.728,47.577,158.946
C08905=1025.246,177.749,386.012,168.724,47.581,158.946
C08906=1025.240,177.500,386.033,168.721,47.586,158.946
C08907=1025.234,177.251,386.056,168.717,47.590,158.947
C08908=1025.228,177.002,386.079,168.713,47.595,158.947
C08909=1025.223,176.754,386.102,168.709,47.599,158.948
C08910=1025.216,176.504,386.124,168.707,47.603,158.948
C08911=1025.211,176.255,386.147,168.703,47.607,158.948
C08912=1025.205,176.007,386.170,168.700,47.612,158.949
C08913=1025.200,175.758,386.192,168.696,47.616,158.949
C08914=1025.194,175.509,386.214,168.692,47.620,158.950
C08915=1025.188,175.260,386.237,168.689,47.625,158.950
C08916=1025.182,175.011,386.260,168.686,47.629,158.950
C08917=1025.176,174.762,386.281,168.682,47.633,158.951
C08918=1025.170,174.513,386.304,168.678,47.638,158.951
C08919=1025.165,174.264,386.327,168.675,47.642,158.952
C08920=1025.159,174.015,386.349,168.672,47.646,158.952
C08921=1025.153,173.767,386.371,168.668,47.651,158.953
C08922=1025.147,173.518,386.394,168.664,47.655,158.953
C08923=1025.142,173.269,386.417,168.661,47.659,158.953
C08924=1025.136,173.020,386.439,168.658,47.663,158.954
C08925=1025.130,172.771,386.462,168.654,47.667,158.954
C08926=1025.124,172.522,386.484,168.651,47.672,158.955
C08927=1025.118,172.239,386.510,168.647,47.677,158.955
C08928=1025.111,171.956,386.535,168.643,47.682,158.955
C08929=1025.105,171.673,386.561,168.639,47.686,158.956
C08930=1025.099,171.390,386.586,168.636,47.691,158.956
C08931=1025.093,171.141,386.608,168.632,47.696,158.957
C08932=1025.087,170.892,386.631,168.628,47.700,158.957
C08933=1025.082,170.643,386.653,168.624,47.704,158.957
C08934=1025.076,170.394,386.676,168.622,47.708,158.958
C08935=1025.070,170.145,386.697,168.618,47.713,158.958
C08936=1025.064,169.896,386.720,168.615,47.717,158.959
C08937=1025.059,169.647,386.742,168.612,47.721,158.959
C08938=1025.053,169.399,386.764,168.608,47.726,158.960
C08939=1025.048,169.149,386.787,168.604,47.730,158.960
C08940=1025.042,168.900,386.810,168.601,47.735,158.960
C08941=1025.037,168.651,386.832,168.598,47.738,158.961
C08942=1025.031,168.403,386.854,168.595,47.743,158.961
C08943=1025.025,168.154,386.876,168.591,47.747,158.962
C08944=1025.020,167.905,386.899,168.588,47.752,158.962
C08945=1025.013,167.655,386.921,168.584,47.756,158.963
C08946=1025.008,167.407,386.943,168.581,47.760,158.963
C08947=1025.003,167.158,386.965,168.578,47.764,158.963
C08948=1024.997,166.909,386.987,168.574,47.768,158.964
C08949=1024.992,166.660,387.010,168.571,47.773,158.964
C08950=1024.986,166.411,387.032,168.568,47.777,158.965
C08951=1024.980,166.162,387.054,168.564,47.782,158.965
C08952=1024.975,165.913,387.076,168.560,47.786,158.965
C08953=1024.969,165.664,387.098,168.558,47.790,158.966
C08954=1024.964,165.415,387.121,168.554,47.794,158.966
C08955=1024.958,165.167,387.143,168.551,47.799,158.967
C08956=1024.953,164.917,387.165,168.548,47.803,158.967
C08957=1024.947,164.668,387.188,168.544,47.807,158.968
C08958=1024.941,164.420,387.209,168.541,47.811,158.968
C08959=1024.936,164.170,387.231,168.538,47.815,158.968
C08960=1024.931,163.922,387.254,168.534,47.820,158.969
C08961=1024.925,163.673,387.275,168.531,47.824,158.969
C08962=1024.919,163.423,387.298,168.528,47.829,158.970
C08963=1024.914,163.175,387.320,168.525,47.832,158.970
C08964=1024.908,162.926,387.342,168.522,47.837,158.970
C08965=1024.903,162.677,387.364,168.518,47.841,158.971
C08966=1024.898,162.427,387.386,168.515,47.846,158.971
C08967=1024.891,162.179,387.408,168.511,47.850,158.972
C08968=1024.886,161.930,387.430,168.509,47.854,158.972
C08969=1024.881,161.681,387.452,168.505,47.858,158.972
C08970=1024.875,161.432,387.474,168.502,47.863,158.973
C08971=1024.870,161.183,387.497,168.499,47.867,158.973
C08972=1024.865,160.934,387.519,168.495,47.871,158.974
C08973=1024.859,160.685,387.540,168.492,47.875,158.974
C08974=1024.853,160.436,387.562,168.489,47.879,158.974
C08975=1024.849,160.187,387.584,168.486,47.884,158.975
C08976=1024.842,159.938,387.607,168.482,47.888,158.975
C08977=1024.837,159.689,387.628,168.480,47.892,158.976
C08978=1024.832,159.440,387.651,168.476,47.897,158.976
C08979=1024.826,159.191,387.672,168.472,47.901,158.977
C08980=1024.821,158.942,387.694,168.470,47.905,158.977
C08981=1024.815,158.693,387.715,168.466,47.910,158.978
C08982=1024.809,158.444,387.737,168.464,47.914,158.978
C08983=1024.803,158.195,387.759,168.460,47.918,158.978
C08984=1024.797,157.946,387.780,168.456,47.923,158.979
C08985=1024.792,157.697,387.802,168.454,47.928,158.979
C08986=1024.786,157.448,387.823,168.450,47.932,158.980
C08987=1024.780,157.199,387.845,168.446,47.937,158.980
C08988=1024.775,156.951,387.866,168.444,47.941,158.981
C08989=1024.770,156.701,387.888,168.440,47.946,158.981
C08990=1024.764,156.452,387.909,168.438,47.950,158.982
C08991=1024.757,156.169,387.934,168.433,47.955,158.982
C08992=1024.751,155.886,387.958,168.430,47.960,158.983
C08993=1024.745,155.602,387.983,168.426,47.965,158.983
C08994=1024.738,155.318,388.008,168.423,47.970,158.984
C08995=1024.732,155.070,388.029,168.419,47.974,158.984
C08996=1024.726,154.820,388.050,168.416,47.979,158.985
C08997=1024.721,154.571,388.071,168.414,47.984,158.985
C08998=1024.715,154.322,388.093,168.410,47.988,158.985
C08999=1024.710,154.073,388.115,168.407,47.992,158.986
C09000=1024.703,153.824,388.136,168.404,47.997,158.986
C09001=1024.698,153.576,388.157,168.401,48.001,158.987
C09002=1024.693,153.326,388.178,168.397,48.006,158.987
C09003=1024.687,153.077,388.200,168.394,48.010,158.988
C09004=1024.682,152.828,388.221,168.391,48.015,158.988
C09005=1024.675,152.579,388.243,168.388,48.019,158.989
C09006=1024.670,152.330,388.264,168.385,48.023,158.989
C09007=1024.664,152.081,388.285,168.382,48.028,158.990
C09008=1024.658,151.832,388.307,168.378,48.033,158.990
C09009=1024.653,151.583,388.327,168.375,48.037,158.990
C09010=1024.647,151.334,388.349,168.372,48.042,158.991
C09011=1024.641,151.085,388.370,168.369,48.046,158.992
C09012=1024.636,150.836,388.391,168.366,48.051,158.992
C09013=1024.630,150.587,388.412,168.363,48.055,158.992
C09014=1024.624,150.338,388.434,168.360,48.059,158.993
C09015=1024.619,150.089,388.454,168.356,48.064,158.993
C09016=1024.612,149.840,388.476,168.354,48.069,158.994
C09017=1024.607,149.591,388.497,168.350,48.073,158.994
C09018=1024.602,149.342,388.518,168.347,48.077,158.995
C09019=1024.595,149.093,388.540,168.344,48.082,158.995
C09020=1024.590,148.844,388.560,168.341,48.087,158.996
C09021=1024.584,148.595,388.582,168.338,48.091,158.996
C09022=1024.579,148.345,388.602,168.335,48.095,158.997
C09023=1024.573,148.097,388.624,168.332,48.100,158.997
C09024=1024.567,147.848,388.645,168.329,48.105,158.998
C09025=1024.562,147.599,388.666,168.325,48.109,158.998
C09026=1024.556,147.349,388.687,168.322,48.113,158.998
C09027=1024.550,147.100,388.708,168.319,48.118,158.999
C09028=1024.545,146.852,388.729,168.316,48.123,158.999
C09029=1024.539,146.602,388.750,168.313,48.127,159.000
C09030=1024.533,146.353,388.771,168.310,48.131,159.000
C09031=1024.528,146.104,388.792,168.307,48.136,159.001
C09032=1024.522,145.854,388.813,168.304,48.141,159.001
C09033=1024.517,145.606,388.834,168.301,48.145,159.002
C09034=1024.511,145.357,388.855,168.298,48.150,159.002
C09035=1024.505,145.108,388.876,168.295,48.155,159.003
C09036=1024.499,144.859,388.896,168.291,48.159,159.003
C09037=1024.494,144.610,388.917,168.289,48.163,159.004
C09038=1024.488,144.360,388.938,168.285,48.168,159.004
C09039=1024.483,144.111,388.959,168.282,48.173,159.005
C09040=1024.477,143.863,388.979,168.280,48.177,159.005
C09041=1024.470,143.613,389.001,168.276,48.182,159.006
C09042=1024.465,143.364,389.021,168.274,48.187,159.006
C09043=1024.460,143.115,389.042,168.270,48.191,159.006
C09044=1024.453,142.866,389.063,168.267,48.195,159.007
C09045=1024.448,142.617,389.083,168.264,48.200,159.008
C09046=1024.443,142.368,389.104,168.261,48.205,159.008
C09047=1024.437,142.119,389.125,168.258,48.209,159.009
C09048=1024.430,141.870,389.145,168.255,48.214,159.009
C09049=1024.425,141.621,389.166,168.252,48.219,159.010
C09050=1024.420,141.372,389.187,168.249,48.222,159.010
C09051=1024.414,141.122,389.208,168.246,48.227,159.010
C09052=1024.408,140.873,389.229,168.243,48.232,159.011
C09053=1024.402,140.625,389.249,168.240,48.237,159.011
C09054=1024.397,140.375,389.269,168.237,48.241,159.012
C09055=1024.391,140.091,389.293,168.234,48.246,159.012
C09056=1024.384,139.808,389.317,168.231,48.251,159.013
C09057=1024.378,139.524,389.341,168.226,48.257,159.013
C09058=1024.371,139.241,389.364,168.223,48.262,159.014
C09059=1024.366,138.992,389.384,168.221,48.267,159.015
C09060=1024.360,138.743,389.405,168.217,48.271,159.015
C09061=1024.354,138.493,389.426,168.214,48.275,159.015
C09062=1024.348,138.244,389.446,168.211,48.280,159.016
C09063=1024.343,137.995,389.466,168.208,48.285,159.017
C09064=1024.338,137.746,389.487,168.205,48.289,159.017
C09065=1024.331,137.496,389.507,168.202,48.294,159.018
C09066=1024.326,137.248,389.529,168.199,48.299,159.018
C09067=1024.320,136.999,389.549,168.197,48.303,159.019
C09068=1024.315,136.750,389.569,168.193,48.308,159.019
C09069=1024.309,136.501,389.590,168.191,48.313,159.020
C09070=1024.303,136.251,389.610,168.188,48.316,159.020
C09071=1024.297,136.002,389.631,168.184,48.321,159.020
C09072=1024.291,135.753,389.651,168.182,48.326,159.021
C09073=1024.286,135.504,389.671,168.178,48.331,159.021
C09074=1024.280,135.255,389.691,168.176,48.335,159.022
C09075=1024.274,135.005,389.712,168.173,48.340,159.022
C09076=1024.268,134.757,389.732,168.170,48.345,159.023
C09077=1024.263,134.508,389.752,168.167,48.349,159.023
C09078=1024.257,134.259,389.772,168.164,48.354,159.024
C09079=1024.252,134.010,389.793,168.161,48.359,159.024
C09080=1024.246,133.761,389.813,168.158,48.363,159.025
C09081=1024.241,133.512,389.833,168.155,48.368,159.025
C09082=1024.234,133.262,389.853,168.152,48.373,159.026
C09083=1024.229,133.012,389.874,168.149,48.377,159.026
C09084=1024.223,132.764,389.894,168.146,48.382,159.027
C09085=1024.218,132.514,389.914,168.143,48.386,159.027
C09086=1024.212,132.266,389.934,168.140,48.391,159.028
C09087=1024.207,132.017,389.955,168.138,48.395,159.028
C09088=1024.201,131.768,389.975,168.134,48.400,159.029
C09089=1024.195,131.518,389.996,168.132,48.405,159.029
C09090=1024.189,131.269,390.016,168.128,48.409,159.030
C09091=1024.183,131.020,390.036,168.126,48.414,159.030
C09092=1024.178,130.771,390.055,168.123,48.419,159.031
C09093=1024.173,130.521,390.076,168.120,48.423,159.031
C09094=1024.167,130.273,390.096,168.117,48.428,159.032
C09095=1024.161,130.023,390.116,168.114,48.433,159.032
C09096=1024.155,129.775,390.136,168.112,48.437,159.033
C09097=1024.150,129.525,390.156,168.108,48.442,159.033
C09098=1024.144,129.276,390.176,168.105,48.447,159.034
C09099=1024.137,129.027,390.196,168.102,48.452,159.034
